# B&R Automation Studio project TD52 (part 101)

#### oilskidCyclic.st
```iecst
(*******************************************************************************
OilSkid	 				Oil Skid (cyclic)

This code is confidential AND proprietary to the INNIO Company.
It may NOT be used in any form, or reproduced in any manner,
without written permission of the INNIO Company.
Copyright, INNIO Company, 2019

Customized modifications: -
------------------------

History:
-------
V3.50	07.01.2014	Tinello 	created
		14.11.2014	Tinello		update TO NEW spezi
V4.x	05.12.2014	Walid Mari 	ported into XT4
V4.03.0	24.06.2015	lettenb.	bT_RelOilSkidPumpC: hy for oiltemp.limit circulation pump added
		18.09.2015				demand oilskid for N2 scavenging + ignition selftest added
		21.10.2015				xTOF_PrelubeDem: lag run time added
V4.05.0	04.04.2017	lettenb.	fast start added
V4.05.1	04.04.2018				bRelEngStart_OilSkid interface prepared for series
V4.05.2	25.04.2018	lettenb.	IN_GC.bOilskidDemSTFS demand for slowturn removed, SWAT920/5
V4.07.0 29.11.2018	lettenb.	preheating temp.limits 30/40->40/50°C
		12.02.2019	lettenb.	2505,3428,3431 depending on oil tank temp. OR oil supply temp.
								2508,3446 enable at engine shutdown
V4.07.1 08.04.2019				OUT_GC.tOilSkid_Heater.Do: bN_EngAct_IsZero removed, heater is active until set temp.is reached(krainz, alessio)
		30.07.2019	lettenb.	error condition for OilSkid: 1031 added, corr.for iCnt_OilSkid_HP_PrErr(safety request, doujak andreas) bu01
V4.10.0	03.08.2020	lettenb.	OUT_interfaces for op_state(bEng_Bloc) added
		14.12.2020	lettenb.	TON,TOF reset added to avoid time overrun, cleanup

Instructions FOR use:
--------------------

Description:
------------

Outstandings:
------------

(*******************************************************************************)
PROGRAM _CYCLIC

	(*----------------------------------------------*)
	(* RESET of alarms and warnings 				*)
	(*----------------------------------------------*)
	bAMM_Lev_OilSkid_Sump_Hi		:= FALSE;

	bAMM_Lev_OilSkid_Tank_Ms 		:= FALSE;
	bAMM_Lev_OilSkid_Tank_Lo 		:= FALSE;
	bAMM_Lev_OilSkid_Tank_LoLo 		:= FALSE;

	bAMM_T_OilSkid_Tank_Ms 			:= FALSE;
	bAMM_T_OilSkid_Tank_Lo 			:= FALSE;

	bAMM_T_OilSkid_Supply_Ms 		:= FALSE;
	bAMM_T_OilSkid_Supply_Lo 		:= FALSE;
	bAMM_T_OilSkid_Supply_Hi 		:= FALSE;

	bAMM_Flow_OilSkid_DE_Ms 		:= FALSE;
	bAMM_Flow_OilSkid_DE_Lo 		:= FALSE;
	bAMM_Flow_OilSkid_DE_Hi 		:= FALSE;

	bAMM_Flow_OilSkid_NDE_Ms 		:= FALSE;
	bAMM_Flow_OilSkid_NDE_Lo 		:= FALSE;
	bAMM_Flow_OilSkid_NDE_Hi 		:= FALSE;

	bAMM_Pr_OilSkid_HP_DE_Ms		:= FALSE;
	bAMM_Pr_OilSkid_HP_DE_Lo 		:= FALSE;

	bAMM_Pr_OilSkid_HP_NDE_Ms		:= FALSE;
	bAMM_Pr_OilSkid_HP_NDE_Lo 		:= FALSE;

	bAMM_OilSkid_PumpC_CB			:= FALSE;
	bAMM_DPr_OilSkid_FiltLP_Hi 		:= FALSE;
	bAMM_DPr_OilSkid_FiltHP_DE_Hi 	:= FALSE;
	bAMM_DPr_OilSkid_FiltHP_NDE_Hi 	:= FALSE;

	bAMM_OilSkid_PumpLP_CB 			:= FALSE;
	bAMM_OilSkid_PumpHP_CB 			:= FALSE;
	bAMM_OilSkid_PumpHP_CB_UPS 		:= FALSE;
	bAMM_OilSkid_Fan_CB 			:= FALSE;
	bAMM_OilSkid_Heater_CB 			:= FALSE;

	bAMM_OilSkid_MCB 				:= FALSE;
	bAMM_OilSkid_AuxV 				:= FALSE;
	bAMM_OilSkid_AuxV_UPS 			:= FALSE;

	(*----------------------------------------------*)
	(* RESET of IO's								*)
	(*----------------------------------------------*)
	OUT_GC.tOilSkid_Fan.Do			:= FALSE;
	OUT_GC.tOilSkid_Heater.Do		:= FALSE;
	OUT_GC.tOilSkid_PumpLP.Do		:= FALSE;
	OUT_GC.tOilSkid_PumpHP.Do		:= FALSE;
	OUT_GC.tOilSkid_PumpHP_UPS.Do	:= FALSE;
	OUT_GC.tOilSkid_PumpHP_Soft.Do	:= FALSE;
	OUT_GC.tOilSkid_PumpC.Do		:= FALSE;

	IF Para.bOilSkid_Exist AND IN_GC.tPB2MM.bParaSetupOk  THEN
		(****************************************************************************************************************************************)
		(* monitoring																															*)
		(****************************************************************************************************************************************)
		xTON_PumpLP_10s(IN:= MM2VIS.bOilSkid_PumpLP_Dem, PT:= T#10s); 								(* LP pump runs for 10 seconds *)
		xTON_PumpHP_5s(IN := MM2VIS.bOilSkid_PumpHP_Dem, PT:= T#5s); 								(* HP pump runs for 5 seconds *)

		(*----------------------------------------------*)
		(* error by DI									*)
		(*----------------------------------------------*)
		bAMM_Lev_OilSkid_Sump_Hi		:=  NOT IN_GC.tLev_OilSkid_Sump_Hi.Di; 										(* G.03-LS-001  *)	(* W3418 *)
		bAMM_DPr_OilSkid_FiltLP_Hi 		:=  NOT IN_GC.tDPr_OilSkid_FiltLP_Hi.Di										(* G.03-PDS-001 *)	(* W2505 *)
										AND 	xTON_PumpLP_10s.Q
										AND   ((bRelMon_T_Supply AND IN_GC.tT_OilSkid_Supply.Ai > 55) OR (bRelMon_T_Tank AND IN_GC.tT_OilSkid_Tank.Ai > 55));

		IF (IN_GC.rN_EngAct < 500 AND IN_GC.rN_EngAct > 100 AND NOT IN_GC.bEng_RPSDem) THEN
			bAMM_DPr_OilSkid_FiltHP_DE_Hi  := NOT IN_GC.tDPr_OilSkid_FiltHP_DE_Hi.Di  AND MM2VIS.bOilSkid_PumpHP_Dem;(* G.03-PDS-002 *) (* W2508 *)
			bAMM_DPr_OilSkid_FiltHP_NDE_Hi := NOT IN_GC.tDPr_OilSkid_FiltHP_NDE_Hi.Di AND MM2VIS.bOilSkid_PumpHP_Dem;(* G.03-PDS-003 *) (* W3446 *)
		END_IF;

		bAMM_OilSkid_PumpLP_CB 			:= NOT IN_GC.tOilSkid_PumpLP_CBOk.Di;															(* W3426 *)
		bAMM_OilSkid_PumpHP_CB 			:= NOT IN_GC.tOilSkid_PumpHP_CBOk.Di;															(* W3433 *)
		bAMM_OilSkid_PumpHP_CB_UPS 		:= NOT IN_GC.tOilSkid_PumpHP_CBOk_UPS.Di;														(* W3434 *)
		bAMM_OilSkid_Fan_CB 			:= NOT IN_GC.tOilSkid_Fan_CBOk.Di; 																(* W3437 *)
		bAMM_OilSkid_Heater_CB 			:= NOT IN_GC.tOilSkid_Heater_CBOk.Di;															(* W3438 *)
		bAMM_OilSkid_PumpC_CB			:= NOT IN_GC.tOilSkid_PumpC_CBOk.Di;															(* W3447 *)

		bAMM_OilSkid_MCB 				:= NOT IN_GC.tOilSkid_MCB.Di;																	(* W3439 *)
		bAMM_OilSkid_AuxV 				:= NOT IN_GC.tOilSkid_AuxV_Ok.Di		AND NOT bAMM_OilSkid_PumpHP_CB  						(* W3440 *)
																				AND NOT bAMM_OilSkid_MCB;
		bAMM_OilSkid_AuxV_UPS 			:= NOT IN_GC.tOilSkid_AuxV_Ok_UPS.Di	AND NOT bAMM_OilSkid_PumpHP_CB_UPS;						(* W3441 *)

			bErr_OilSkid_NoVoltage		:= bAMM_OilSkid_MCB OR bAMM_OilSkid_AuxV;

		(*----------------------------------------------*)
		(* error by measurement signal failure 			*)
		(*----------------------------------------------*)
		bAMM_Lev_OilSkid_Tank_Ms	:= Para.bLev_OilSkid_Tank_Exist 	AND NOT IN_GC.tLev_OilSkid_Tank.GoodQual;						(* W3419 *)
		bAMM_T_OilSkid_Tank_Ms		:= Para.bT_OilSkid_Tank_Exist 		AND NOT IN_GC.tT_OilSkid_Tank.GoodQual;							(* W3421 *)
		bAMM_T_OilSkid_Supply_Ms	:= Para.bT_OilSkid_Supply_Exist 	AND NOT IN_GC.tT_OilSkid_Supply.GoodQual;						(* W3423 *)
		bAMM_Flow_OilSkid_DE_Ms		:= Para.bFlow_OilSkid_DE_Exist 		AND NOT IN_GC.tFlow_OilSkid_DE.GoodQual;						(* W3427 *)
		bAMM_Flow_OilSkid_NDE_Ms	:= Para.bFlow_OilSkid_NDE_Exist 	AND NOT IN_GC.tFlow_OilSkid_NDE.GoodQual;						(* W3430 *)
		bAMM_Pr_OilSkid_HP_DE_Ms	:= Para.bPr_OilSkid_HP_DE_Exist 	AND NOT IN_GC.tPr_OilSkid_HP_DE.GoodQual;						(* W3435 *)
		bAMM_Pr_OilSkid_HP_NDE_Ms	:= Para.bPr_OilSkid_HP_NDE_Exist 	AND NOT IN_GC.tPr_OilSkid_HP_NDE.GoodQual;						(* W3442 *)

			(* Release monitoring	*)
			xTOF_AMM_Lev_Tank_Ms(IN := bAMM_Lev_OilSkid_Tank_Ms, 	PT:= T#10s);	(* TOF because of filtered signals *)
			xTOF_AMM_T_Tank_Ms(IN 	:= bAMM_T_OilSkid_Tank_Ms, 	 	PT:= T#10s);
			xTOF_AMM_T_Supply_Ms(IN := bAMM_T_OilSkid_Supply_Ms, 	PT:= T#10s);
			xTOF_AMM_Flow_DE_Ms(IN 	:= bAMM_Flow_OilSkid_DE_Ms, 	PT:= T#10s);
			xTOF_AMM_Flow_NDE_Ms(IN := bAMM_Flow_OilSkid_NDE_Ms, 	PT:= T#10s);
			xTOF_Pr_HP_DE_Ms(IN 	:= bAMM_Pr_OilSkid_HP_DE_Ms,	PT:= T#10s);
			xTOF_Pr_HP_NDE_Ms(IN 	:= bAMM_Pr_OilSkid_HP_NDE_Ms,	PT:= T#10s);

			bRelMon_Lev_Tank		:= Para.bLev_OilSkid_Tank_Exist		AND NOT xTOF_AMM_Lev_Tank_Ms.Q;
			bRelMon_T_Tank			:= Para.bT_OilSkid_Tank_Exist		AND NOT xTOF_AMM_T_Tank_Ms.Q;
			bRelMon_T_Supply		:= Para.bT_OilSkid_Supply_Exist		AND NOT xTOF_AMM_T_Supply_Ms.Q;
			bRelMon_Flow_DE			:= Para.bFlow_OilSkid_DE_Exist		AND NOT xTOF_AMM_Flow_DE_Ms.Q;
			bRelMon_Flow_NDE		:= Para.bFlow_OilSkid_NDE_Exist		AND NOT xTOF_AMM_Flow_NDE_Ms.Q;
			bRelMon_Pr_HP_DE		:= Para.bPr_OilSkid_HP_DE_Exist		AND NOT xTOF_Pr_HP_DE_Ms.Q;
			bRelMon_Pr_HP_NDE		:= Para.bPr_OilSkid_HP_NDE_Exist	AND NOT xTOF_Pr_HP_NDE_Ms.Q;

		(*----------------------------------------------*)
		(* error by level 		 						*)
		(*----------------------------------------------*)
		xGR_MINR_Lev_OilSkid_Tank(In:= IN_GC.tLev_OilSkid_Tank.Ai, Gw:= Para.rLev_OilSkid_Tank_LoLo, Hy:= 0.05);	(* 5% hysteresis *)

		bAMM_Lev_OilSkid_Tank_LoLo	:= xGR_MINR_Lev_OilSkid_Tank.Q 								AND bRelMon_Lev_Tank;					(* A2208 *)
		bAMM_Lev_OilSkid_Tank_Lo	:= (IN_GC.tLev_OilSkid_Tank.Ai < Para.rLev_OilSkid_Tank_Lo) AND bRelMon_Lev_Tank;					(* W3420 *)

		(*----------------------------------------------*)
		(* error by temperature	 						*)
		(*----------------------------------------------*)
		bAMM_T_OilSkid_Tank_Lo 		:= (IN_GC.tT_OilSkid_Tank.Ai   < 20) AND bOMSS_MAT AND bRelMon_T_Tank;								(* W3422 *)

		bAMM_T_OilSkid_Supply_Lo	:= (IN_GC.tT_OilSkid_Supply.Ai < Para.rT_OilSkid_Supply_Lo)	AND bRelMon_T_Supply					(* W3424 *)
																								AND MM2VIS.bOilSkid_PumpLP_Dem
																								AND bEng_Run_30m;

		bAMM_T_OilSkid_Supply_Hi	:= (IN_GC.tT_OilSkid_Supply.Ai > Para.rT_OilSkid_Supply_Hi)	AND bRelMon_T_Supply
																								AND MM2VIS.bOilSkid_PumpLP_Dem;			(* W3425 *)

		(*----------------------------------------------*)
		(* error by flow		 						*)
		(*----------------------------------------------*)
		IF (bRelMon_T_Supply AND IN_GC.tT_OilSkid_Supply.Ai > 55) OR 			(* tank   temperature > 55°C *)
		   (bRelMon_T_Tank   AND IN_GC.tT_OilSkid_Tank.Ai   > 55) THEN 			(* supply temperature > 55°C *)
			bErr_Flow_OilSkid_DE_Lo		:= (IN_GC.tFlow_OilSkid_DE.Ai  < Para.rFlow_OilSkid_DE_Lo);
			bErr_Flow_OilSkid_NDE_Lo	:= (IN_GC.tFlow_OilSkid_NDE.Ai < Para.rFlow_OilSkid_NDE_Lo);
		ELSE
			bErr_Flow_OilSkid_DE_Lo		:= (IN_GC.tFlow_OilSkid_DE.Ai  < 4);	(* 4 l/min *)
			bErr_Flow_OilSkid_NDE_Lo	:= (IN_GC.tFlow_OilSkid_NDE.Ai < 4);	(* 4 l/min *)
		END_IF;

		bAMM_Flow_OilSkid_DE_Lo		:= bErr_Flow_OilSkid_DE_Lo	AND xTON_PumpLP_10s.Q			AND bRelMon_Flow_DE;					(* W3428 *)
		bAMM_Flow_OilSkid_NDE_Lo	:= bErr_Flow_OilSkid_NDE_Lo	AND xTON_PumpLP_10s.Q			AND bRelMon_Flow_NDE;					(* W3431 *)

		bAMM_Flow_OilSkid_DE_Hi		:= (IN_GC.tFlow_OilSkid_DE.Ai  > Para.rFlow_OilSkid_DE_Hi)	AND bRelMon_Flow_DE;					(* W3429 *)
		bAMM_Flow_OilSkid_NDE_Hi	:= (IN_GC.tFlow_OilSkid_NDE.Ai > Para.rFlow_OilSkid_NDE_Hi)	AND bRelMon_Flow_NDE;					(* W3432 *)

		(*----------------------------------------------*)
		(* error by pressure	 						*)
		(*----------------------------------------------*)
			(* oil pressure in high pressure circuit OK *)
			bPr_OilSkid_HP_DE_Ok	:= IN_GC.tPr_OilSkid_HP_DE.Ai  > Para.rPr_OilSkid_HP_Lo;
			bPr_OilSkid_HP_NDE_Ok	:= IN_GC.tPr_OilSkid_HP_NDE.Ai > Para.rPr_OilSkid_HP_Lo;

			(* release by stable oil pressure *)
			xTON_PressOK_2s(IN:= ((bPr_OilSkid_HP_DE_Ok  AND bRelMon_Pr_HP_DE)  OR NOT Para.bPr_OilSkid_HP_DE_Exist ) AND
								 ((bPr_OilSkid_HP_NDE_Ok AND bRelMon_Pr_HP_NDE) OR NOT Para.bPr_OilSkid_HP_NDE_Exist) AND
								 (Para.bPr_OilSkid_HP_DE_Exist OR Para.bPr_OilSkid_HP_NDE_Exist),		(* at least on sensor exist *)
							PT:= T#2s);
			bRel_OilSkid_Pr	  := xTON_PressOK_2s.Q;

		bAMM_Pr_OilSkid_HP_DE_Lo 	:= NOT bPr_OilSkid_HP_DE_Ok	 AND xTON_PumpHP_5s.Q AND bRelMon_Pr_HP_DE;								(* W3436 *)
		bAMM_Pr_OilSkid_HP_NDE_Lo 	:= NOT bPr_OilSkid_HP_NDE_Ok AND xTON_PumpHP_5s.Q AND bRelMon_Pr_HP_NDE;							(* W3443 *)

		(****************************************************************************************************************************************)
		(* control																																*)
		(****************************************************************************************************************************************)
		xTOF_NoSpeed_30s(IN:= NOT bN_EngAct_IsZero, PT:= T#30s);							(* engine is running *)

			(*----------------------------------------------*)
			(* preheating		 							*)
			(*----------------------------------------------*)
			IF bRelMon_T_Tank AND bOMSS_MAT THEN
				IF 		IN_GC.tT_OilSkid_Tank.Ai >= 50 	THEN   bOilSkid_Heater	:= FALSE;
				ELSIF 	IN_GC.tT_OilSkid_Tank.Ai <  40 	THEN   bOilSkid_Heater	:= TRUE; 	END_IF;

				OUT_GC.tOilSkid_Heater.Do	:=	bOilSkid_Heater
										AND NOT bAMM_OilSkid_Heater_CB
										AND NOT bErr_OilSkid_NoVoltage
										AND NOT IN_GC.bMsg1031
										AND NOT IN_GC.bMsg1054;
			END_IF;

			(*----------------------------------------------*)
			(* Service										*)
			(*----------------------------------------------*)
			IF 		NOT M_DREHZ							(* engine is not running *)
				AND NOT bAMM_Lev_OilSkid_Sump_Hi
				AND NOT IN_GC.bEng_RPSDem				(* engine is not demanded *)
				AND    (IN_GC.tT_OilSkid_Tank.Ai >= 20) (* oil temperature OK *)
				AND     bRelMon_T_Tank  THEN

				(* oilskid oil high pressure pump runtime *)
				xTON_PumpHP_DemOn(IN:= bPumpHP_DemService, PT:= Para.tiOilSkid_PumpHP_Run);

				IF 	IN_GC.tOilSkid_PumpHP_DemOn.Di AND NOT xTOF_NoSpeed_30s.Q			THEN bPumpHP_DemService	:= TRUE; 	END_IF;
				IF (IN_GC.tOilSkid_PumpHP_DemOff.Di OR xTON_PumpHP_DemOn.Q) 			THEN bPumpHP_DemService	:= FALSE;	END_IF;

				(* reset if pump isn't running *)
				IF (xTON_PumpHP_DemOn.ET > T#5s) AND NOT MM2VIS.bOilSkid_PumpHP_Dem 	THEN bPumpHP_DemService	:= FALSE;	END_IF;

				(* demand oilskid oil high pressure pump for N2 or IgnSelfTest *)//SWAT920/5
				xTOF_PrelubeDem(IN:= IN_GC.bN2_ScavCoPrelubeOn OR IN_GC.bEO_PrelubeDemIgn, PT:= T#60s);(* lag run time / until engine stand still *)//SWAT920/5
				bPumpHP_DemN2Ign := xTOF_PrelubeDem.Q;

			ELSE
				xTON_PumpHP_DemOn(IN:= FALSE, PT:= T#0s);
				xTOF_PrelubeDem  (IN:= FALSE, PT:= T#0s);

				bPumpHP_DemService 	:= FALSE;
				bPumpHP_DemN2Ign	:= FALSE;
			END_IF;

			OUT_GC.bRelEngTurn_OilSkid	:= bRel_OilSkid_Pr AND(bPumpHP_DemService OR bPumpHP_DemN2Ign);	(* release engine turn *)

			(*----------------------------------------------*)
			(* release engine operation						*)
			(*----------------------------------------------*)
			IF    IN_GC.bEng_RPSDem AND (IN_GC.tT_OilSkid_Tank.Ai >= 20)
			THEN
				bPumpHP_DemEngOp			:= (IN_GC.rN_EngAct < 500);
				OUT_GC.tOilSkid_PumpLP.Do	:= (IN_GC.rN_EngAct > 200)
										AND NOT bAMM_OilSkid_PumpLP_CB
										AND NOT bErr_OilSkid_NoVoltage
										AND NOT IN_GC.bMsg1031
										AND NOT IN_GC.bMsg1054;
			ELSE
				bPumpHP_DemEngOp 		:= FALSE;
			END_IF;

			OUT_GC.bRelEngOp_OilSkid	:= bRel_OilSkid_Pr AND bPumpHP_DemEngOp;	(* release engine operation *)
			OUT_GC.bRelEngStart_OilSkid	:= NOT bAMM_T_OilSkid_Tank_Lo AND NOT bAMM_Lev_OilSkid_Tank_LoLo; (* oilskid ready for fast start *)

			(*----------------------------------------------*)
			(* cooling										*)
			(*----------------------------------------------*)
			IF NOT bN_EngAct_IsZero THEN

				IF 	bRelMon_T_Tank THEN
					IF 	  IN_GC.tT_OilSkid_Tank.Ai   >  Para.rT_OilSkid_Tank_Set 		THEN  bOilSkid_Fan	:= TRUE;
					ELSIF IN_GC.tT_OilSkid_Tank.Ai   < (Para.rT_OilSkid_Tank_Set - 5)	THEN  bOilSkid_Fan	:= FALSE; 	END_IF;

				ELSIF bRelMon_T_Supply 	THEN				(* switch to supply temperature in case of tank temp. error *)
					IF 	  IN_GC.tT_OilSkid_Supply.Ai >  Para.rT_OilSkid_Tank_Set 		THEN  bOilSkid_Fan	:= TRUE;
					ELSIF IN_GC.tT_OilSkid_Supply.Ai < (Para.rT_OilSkid_Tank_Set - 5) 	THEN  bOilSkid_Fan	:= FALSE; 	END_IF;
				END_IF;

				OUT_GC.tOilSkid_Fan.Do	:=	bOilSkid_Fan
									AND NOT bAMM_OilSkid_Fan_CB
									AND NOT bErr_OilSkid_NoVoltage
									AND NOT IN_GC.bMsg1031
									AND NOT IN_GC.bMsg1054;
			END_IF;

			(*----------------------------------------------*)
			(* circulation pump								*)
			(*----------------------------------------------*)
			IF 	  IN_GC.tT_OilSkid_Tank.Ai >= 22.0 THEN bT_RelOilSkidPumpC := TRUE;
			ELSIF IN_GC.tT_OilSkid_Tank.Ai <  20.0 THEN bT_RelOilSkidPumpC := FALSE; END_IF;

			OUT_GC.tOilSkid_PumpC.Do :=   ((MM2VIS.bOilSkid_Heater_Dem AND bT_RelOilSkidPumpC) OR (IN_GC.rN_EngAct > 200)) 	(* Heater is running *)
									AND	NOT bAMM_OilSkid_PumpC_CB
									AND NOT bErr_OilSkid_NoVoltage
									AND NOT IN_GC.bMsg1031
									AND NOT IN_GC.bMsg1054;

			(*----------------------------------------------*)
			(* engine stop									*)
			(*----------------------------------------------*)
			IF 	NOT IN_GC.bEng_RPSDem AND xTOF_NoSpeed_30s.Q THEN
				bPumpHP_DemEngStop			:= (IN_GC.rN_EngAct < 500);
				OUT_GC.tOilSkid_PumpLP.Do	:=	NOT bRel_OilSkid_Pr
											AND NOT bAMM_OilSkid_PumpLP_CB
											AND NOT bErr_OilSkid_NoVoltage
											AND NOT IN_GC.bMsg1031
											AND NOT IN_GC.bMsg1054;
				xTON_PumpHP_Dem_5s(IN := bPumpHP_DemEngStop, PT:= T#5s);	 			(* HP pump demand for 5 seconds *)

				IF  NOT bRel_OilSkid_Pr AND	EDGEPOS(xTON_PumpHP_Dem_5s.Q) THEN
					VIS2MM.iCnt_OilSkid_HP_PrErr := VIS2MM.iCnt_OilSkid_HP_PrErr + 1; 	(* Perm: error counter for high pressure *)
				END_IF;
			ELSE
				xTON_PumpHP_Dem_5s(IN:= FALSE, PT:= T#0s);
				bPumpHP_DemEngStop := FALSE;
			END_IF;

			(*----------------------------------------------*)
			(* engine faststart								*)
			(*----------------------------------------------*)
			xTON_FS(IN:= (IN_GC.rN_EngAct > 0), PT:= T#4s);
			IF 	IN_GC.bEng_Start THEN
				IF  NOT bRel_OilSkid_Pr AND	EDGEPOS(xTON_FS.Q) THEN
					VIS2MM.iCnt_OilSkid_HP_PrErr := VIS2MM.iCnt_OilSkid_HP_PrErr + 1; 	(* Perm: error counter for high pressure *)
				END_IF;
			END_IF;

			(*----------------------------------------------*)
			(* high pressure pump / UPS						*)
			(*----------------------------------------------*)
			xTOF_PumpHP_Dem(IN:= bPumpHP_DemService OR bPumpHP_DemN2Ign OR bPumpHP_DemEngOp OR bPumpHP_DemEngStop, PT:= T#1s);

			OUT_GC.tOilSkid_PumpHP_Soft.Do	:= xTOF_PumpHP_Dem.Q AND NOT IN_GC.bMsg1031
																 AND NOT IN_GC.bMsg1054;

			OUT_GC.tOilSkid_PumpHP.Do		:= xTOF_PumpHP_Dem.Q AND NOT xTOF_PumpHP_UPS.Q
																 AND NOT bAMM_OilSkid_PumpHP_CB
																 AND NOT bErr_OilSkid_NoVoltage
																 AND NOT IN_GC.bMsg1031
																 AND NOT IN_GC.bMsg1054;

			xTOF_PumpHP(IN:= OUT_GC.tOilSkid_PumpHP.Do, PT:= T#1s);

			OUT_GC.tOilSkid_PumpHP_UPS.Do	:= xTOF_PumpHP_Dem.Q AND NOT xTOF_PumpHP.Q
																 AND NOT bAMM_OilSkid_PumpHP_CB_UPS
																 AND NOT bAMM_OilSkid_AuxV_UPS
																 AND     xTOF_NoSpeed_30s.Q			(* demand only if shutdown *)
																 AND NOT IN_GC.bMsg1031
																 AND NOT IN_GC.bMsg1054;
			xTOF_PumpHP_UPS(IN:= OUT_GC.tOilSkid_PumpHP_UPS.Do, PT:= T#1s);

		IF 		IN_GC.bMsg1031  													(* A1031 emergency stop *)
			OR  IN_GC.bMsg1054  													(* A1054 fire alarm *)
			OR (MM2VIS.bMsg2208  AND NOT bMsg2208_Test) 							(* A2208 oilskid tank level minimum *)
			OR (bAMM_OilSkid_MCB AND     bN_EngAct_IsZero) THEN						(* W3439 Oilskid main switch auxiliaries opened *)

			bPumpHP_DemService 			:= FALSE;									(* NO demand of high pressure pump 	 *)
			bPumpHP_DemN2Ign			:= FALSE;									(* NO demand of high pressure pump 	 *)
			bPumpHP_DemEngOp			:= FALSE;									(* NO demand of high pressure pump 	 *)
			OUT_GC.bRelEngOp_OilSkid 	:= FALSE;									(* NO release of engine operation 	 *)
			OUT_GC.bRelEngTurn_OilSkid	:= FALSE;									(* NO release of engine barring gear *)
			OUT_GC.bRelEngStart_OilSkid	:= FALSE; 									(* NO oilskid ready for fast start   *)
		END_IF;

	ELSE (* inactive OilSkid *)
		xTON_PumpLP_10s(IN:= FALSE, PT:= T#0s);
		xTON_PumpHP_5s(IN:= FALSE, PT:= T#0s);
		xTON_PressOK_2s(IN:= FALSE, PT:= T#0s);
		xTON_PumpHP_DemOn(IN:= FALSE, PT:= T#0s);
		xTON_PumpHP_Dem_5s(IN:= FALSE, PT:= T#0s);
		xTON_FS(IN:= FALSE, PT:= T#0s);

		xTOF_NoSpeed_30s(IN:= FALSE, PT:= T#0s);
		xTOF_PrelubeDem(IN:= FALSE, PT:= T#0s);
		xTOF_PumpHP_UPS(IN:= FALSE, PT:= T#0s);
		xTOF_PumpHP(IN:= FALSE, PT:= T#0s);

		bPumpHP_DemService			:= FALSE;										(* NO demand of high pressure pump 	 *)
		bPumpHP_DemN2Ign			:= FALSE;										(* NO demand of high pressure pump 	 *)
		bPumpHP_DemEngOp			:= FALSE;										(* NO demand of high pressure pump 	 *)
		bPumpHP_DemEngStop			:= FALSE;										(* NO demand of high pressure pump 	 *)
		OUT_GC.bRelEngOp_OilSkid 	:= TRUE;										(*    release engine operation  	 *)
		OUT_GC.bRelEngTurn_OilSkid	:= TRUE;										(*    release engine barring gear	 *)
		OUT_GC.bRelEngStart_OilSkid	:= TRUE; 										(*    oilskid ready for fast start   *)
	END_IF;

	OUT_GC.bAMM_OilSkid_PumpLP_CB := bAMM_OilSkid_PumpLP_CB;						(* bEng_Bloc *)
	OUT_GC.bAMM_OilSkid_PumpHP_CB := bAMM_OilSkid_PumpHP_CB;						(* bEng_Bloc *)
	OUT_GC.bAMM_OilSkid_MCB       := bAMM_OilSkid_MCB;								(* bEng_Bloc *)

END_PROGRAM
```

#### oilskid.var
```iecst
VAR
	bErr_Flow_OilSkid_DE_Lo : BOOL := FALSE; (*Internal WARNING: OilSkid oil flow to DE - low*)
	bErr_Flow_OilSkid_NDE_Lo : BOOL := FALSE; (*Internal WARNING: OilSkid oil flow to NDE - low*)
	bErr_OilSkid_NoVoltage : BOOL := FALSE; (*Internal WARNING: OilSkid NO Voltage*)
	bOilSkid_Fan : BOOL := FALSE; (*Fan*)
	bOilSkid_Heater : BOOL := FALSE; (*Heater*)
	bPr_OilSkid_HP_DE_Ok : BOOL := FALSE; (*Oil pressure in high pressure circuit to DE bearing OK*)
	bPr_OilSkid_HP_NDE_Ok : BOOL := FALSE; (*Oil pressure in high pressure circuit to NDE bearing OK*)
	bPumpHP_DemEngOp : BOOL := FALSE; (*Demand high pressure pump for engine operation *)
	bPumpHP_DemEngStop : BOOL := FALSE; (*Demand high pressure pump for engine stop*)
	bPumpHP_DemService : BOOL := FALSE; (*Demand high pressure pump for service*)
	bPumpHP_DemN2Ign : BOOL := FALSE; (*Demand high pressure pump for N2 or IgnSelfTest*)
	bRelMon_Lev_Tank : BOOL := FALSE; (*Release monitoring OilSkid tank level*)
	bRelMon_Pr_HP_DE : BOOL := FALSE; (*Release monitoring OilSkid oil pressure in high pressure circuit to DE bearing*)
	bRelMon_Pr_HP_NDE : BOOL := FALSE; (*Release monitoring OilSkid oil pressure in high pressure circuit to NDE bearing*)
	bRelMon_T_Supply : BOOL := FALSE; (*Release monitoring OilSkid supply temperature*)
	bRelMon_T_Tank : BOOL := FALSE; (*Release monitoring OilSkid tank temperature*)
	bRel_OilSkid_Pr : BOOL := FALSE; (*Release by oil pressure*)
	bT_RelOilSkidPumpC : BOOL := FALSE; (*Release circ.pump by oil temperature*)
	xGR_MINR_Lev_OilSkid_Tank : GR_MINR := (0);
	xTOF_AMM_Flow_DE_Ms : TOF := (0);
	xTOF_AMM_Flow_NDE_Ms : TOF := (0);
	xTOF_AMM_Lev_Tank_Ms : TOF := (0);
	xTOF_AMM_T_Supply_Ms : TOF := (0);
	xTOF_AMM_T_Tank_Ms : TOF := (0);
	xTOF_NoSpeed_30s : TOF := (0);
	xTOF_Pr_HP_DE_Ms : TOF := (0);
	xTOF_Pr_HP_NDE_Ms : TOF := (0);
	xTOF_PumpHP : TOF := (0);
	xTOF_PumpHP_Dem : TOF := (0);
	xTOF_PumpHP_UPS : TOF := (0);
	xTON_PressOK_2s : TON := (0);
	xTON_PumpHP_5s : TON := (0);
	xTON_PumpHP_DemOn : TON := (0);
	xTON_PumpLP_10s : TON := (0);
	xTOF_PrelubeDem : TOF;
	xTON_FS : TON := (0);
	xTON_PumpHP_Dem_5s : TON := (0);
END_VAR
```

### Program Logical/Generator/PermGC (IEC, version 4.09.0) - + PermanentMemory

- PermGCCyclic.st (not readable text: treated as protected, skipped)

- PermGCInit.st (not readable text: treated as protected, skipped)

#### PermGC.var
```iecst
VAR
	pm_Error : UINT;
	write_once : BOOL;
	pm_len : UDINT;
	ModulName : STRING[35];
	DatObjInfo_01 : DatObjInfo;
	pm_id : UDINT;
	pm_p : UDINT;
	bCreateDataObj : BOOL;
	perm_par_vers : UINT;
	DatObjRead_01 : DatObjRead;
	DatObjDelete_PermMem : DatObjDelete;
	DatObjCreate_01 : DatObjCreate;
	DatObjWrite_01 : DatObjWrite;
	ulChecksumOld : UDINT;
	ulPMPointer : UDINT;
	ulChkValue : UDINT;
	TON_WritePMEM : TON;
	ulChecksum : UDINT;
	bWriteDataObj : BOOL;
	TON_WarnDelay : TON;
	TON_BlockMinFileAge : TON; (*waiting time without file write after successful performed write*)
	bBlock_MinFileAge : BOOL := FALSE; (*pause the perm file write after each sucessful write*)
	iPM_WriteCnt : UDINT; (* *) (*old VarName: usPMWriteCnt*)
END_VAR
VAR CONSTANT
	ERR_NOERROR : UINT := 0;
END_VAR
VAR
	pmm : Perm_GC_Struct;
END_VAR
```

### Program Logical/Generator/MsgGC (IEC, version 4.14.0) - messages

#### MsgGCCyclic.st
```iecst
(*******************************************************************************
MsgGC	 			 alarms generation MM_generator

This code is confidential and proprietary to the INNIO Company.
It may not be used in any form, or reproduced in any manner,
without written permission of the INNIO Company.
Copyright, INNIO Company, 2025

Customized modifications: -
------------------------

History:
-------
V0.01.0	02.11.2011	lettenb.	new
V0.01.0	22.04.2013	Denk		xMsg3319.Prio := 3; 	deleted (Copy-paste failure)
		27.05.2013	Lettenb.	reset OUT_xx.txx2AB.bGnlTripx changed
V0.02.0 21.06.2013	Zengerer	W3566 added
V4.00.0 04.03.2014	lettenb.	logger added
V4.00.1	19.05.2014	lettenb.	3566 bugfix
		30.05.2014				1037 prio4 -> 2, bugfix
V4.00.2	09.12.2014				1036.Enable := TRUE -> IN_GC.tPB2MM.bSys_Run(920 stapelfeld)
								1110 Aktivierung bei BR9 wenn n_nenn 20sec > 750rpm für (Einfahrprogramm 500rpm)(920 stapelfeld)
								1126,2277 bei BR9 nur aktiv wenn n_nenn > 750rpm	(wegen Einfahrprogramm)(920 stapelfeld)
								2202,2203,2204,2205,2206,2207,2502,2503,2504,2631,2632,2633,2634,2637 added (920)
V4.03.0	22.07.2015	lettenb.	1038,1073,1109,1110,1111,1112,1126,1127,1143,1144 modif. 2690,2691,3393 new, dyn.gridcode III(thaler)
								_TC2 var.removed(bugfix vvm maping failure)
V4.04.0	10.05.2016	lettenb.	1127 monitoring activation acc.specification(kru) removed(bU_Gen_Mon_Ena)
								3468 added(T_GenAirIn2)
		23.02.2017				3440 TON 2s hinzu, unterdrückung 3440 bei wiedereinschaltung hauptschalter/schutzschalter
		28.07.2017	502423184	A2202 AND A2203 disabled due TO SWAT 920 # 3
V4.05.0	06.12.2017	lettenb.	W3566 disabled(->3593/update gridcode functions)
								2316 added, 2277 bMMD_GenAlarmTestOn added, grid code logic(thaler)
		09.04.2018				1036 bParaSetupOk added to avoid alarm at plc startup, bugfix
V4.07.0	19.10.2018	lettenb.	3468 bParaSetupOk added to avoid alarm at plc startup, bugfix
		29.11.2018	lettenb.	2505 delay 10s->120s,3428 delay 120s, 3431 delay 120s, 2998 added
		15.02.2019	lettenb.	3429,3432 delay 0s->120s
		04.03.2019	lettenb.	1038,1144 IN_GC.tP_GenRev_Ext.Di / IN_GC.tI_GenAsy_Ext.Di - DIs act directly on alarms without delay
V4.07.1	04.06.2019	lettenb.	2336 added, 3573 disabled
V4.09.0	02.12.2019	lettenb.	9311 added, acc.VDE-AR-N 4110 / 10.2.3.1(thaler), protection test mapping
		03.02.2020	lettenb.	2156,2157,2998 write max.1x per minute, bugfix
		04.05.2020	lettenb.	xTON_SecTick added for cycle time undependency, bugfix
V4.10.0	22.12.2020	lettenb.	1112: RiskClass setting corr.acc.TI 1100-0111
V4.11.0	25.01.2020	MayerR		9285,9351 added, voltage droop, tU_SetExt_Norm -> tU_SetExtAI_Norm renamed
V4.12.0	21.11.2022	lettenb.	9365,9366,9367,9368 added, automatic bearing greasing system
								1109,1110: avoid alarm during gen.dexcitation and gcb closing to dead bb(DUB15 BF43),#912
		19.12.2022	Perktold	added comments for sr-code (EN 13849-1 / 4.6.3) for A1038
V4.13.0	12.06.2023	Rimal		2371 and 2372 added, oilskid
		04.07.2023	Perktold	A2373 and W9372 added, earth fault protection via MMD signals
V4.14.0	17.10.2024	Theobald	Alarm 1112,1121,1122,1123,1124,1125,1143,1144 priority changed from 2 to 3 (2024-223)
		25.10.2024	Farre		Reverse power status OUT_GC.bPact_Rev to SY (2024-241)
		18.11.2024	Farre		Enable "unbalance current monitoring A1144" based on Para.bCAsym_Ena (2024-234)
		04.03.2025	Perktold	Alarm 1144 priority changed back to 2 (from 3)

Instructions for use:
--------------------
1) declare alarm with function block "Alm"
	declare buffert alarm bit MM2VIS.bMsg<message number>

2) use template to create a new alarm,
   substitue 0000 by alarm number and make settings:

	xMsg0000.Enable		:=	TRUE;		enable/disable alarm
	xMsg0000.Set		:=	FALSE;		alarm set condition
	xMsg0000.PT			:=	T#0s;		alarm delay time
	xMsg0000.Prio		:=	1;			alarm priority: 1-3 = trip, 4 = warning
	xMsg0000.RiskClass	:=	3;			risk class for remote alarm reset
	xMsg0000.Reset		:=	FALSE;		FALSE: for all standard alarms	prio 1,2,3 and warnings prio 4
										TRUE : for autoreset alarms

	MM2VIS.bMsg0000			:=	xMsg0000.Q;	connect buffert alarm bit for VIS and control

3)  expand INIT

Outstandings:
------------
sort msg by number
(*******************************************************************************)
PROGRAM _CYCLIC

	(* reset general trip *)
	OUT_GC.tGC2AB.bGnlTrip1		:=	FALSE;
	OUT_GC.tGC2AB.bGnlTrip2		:=	FALSE;
	OUT_GC.tGC2AB.bGnlTrip3		:=	FALSE;
	OUT_GC.tGC2AB.bGnlWarning	:=	FALSE;
	OUT_GC.tGC2AB.bTriptype1	:=	FALSE;
	OUT_GC.tGC2AB.bTriptype2	:=	FALSE;
	OUT_GC.tGC2AB.bTriptype3	:=	FALSE;

	(*------------------------------------------------------------------------------*)
	xGR_MAX_M_D_1400(In := IN_GC.rN_EngAct,Gw := Para.rN_EngNom - 100.0, Hy := 10);
	M_D1400 := xGR_MAX_M_D_1400.Q AND IN_GC.tPB2MM.bParaSetupOk;

	xTON_FG_GENUW(IN := M_D1400 AND NOT IN_GC.tGenDeexitDem.Do, PT := T#20s);
	bU_Gen_Mon_Ena := xTON_FG_GENUW.Q;

	xTON_Eng_Run_10s(IN := IN_GC.tEng_Run.Do , PT := T#10s);
	bEng_Run_10s := xTON_Eng_Run_10s.Q;

	xTON_Eng_Run_20s(IN := IN_GC.tEng_Run.Do , PT := T#20s);
	bEng_Run_20s := xTON_Eng_Run_20s.Q;

	xGR_MAXR_M_HDREHZ(In := IN_GC.rN_EngAct , Gw := Para.rN_EngStart_LimHiHi, Hy := Para.rN_EngStart_HyHiHi );
	M_HDREHZ := xGR_MAXR_M_HDREHZ.Q AND IN_GC.tPB2MM.bParaSetupOk;

	xTON_AT24.IN := (IN_GC.tGCB_On.Di OR M_HDREHZ) AND (IN_GC.tEng_Run.Do OR (NOT IN_GC.tEng_SUExc_Rel.Di));
	xTON_AT24.PT := Para.tiP_Gen_Reverse;
	xTON_AT24();
	bP_Gen_Reverse := xTON_AT24.Q;

	xTP_RLSG_W.IN := IN_GC.bEng_Dem_EPS;
	xTP_RLSG_W.PT := Para.tiP_Reverse_Mon_Ena;
	xTP_RLSG_W();
	bP_Reverse_Mon_Ena := xTP_RLSG_W.Q;

	(* A1036 Generator overload/short circuit *)
	xMsg1036.Enable    := IN_GC.tPB2MM.bParaSetupOk;
	xMsg1036.Set       := NOT IN_GC.tOlShortCirc.Di;
	xMsg1036.PT        := T#0s;
	xMsg1036.RiskClass := 4;
	xMsg1036.Prio      := 2;
	xMsg1036.Reset     := FALSE;
	xMsg1036();
	OUT_GC.bMsg1036    := xMsg1036.Q;
	MM2VIS.bMsg1036    := xMsg1036.Q;

	(* A1037 generator winding temperature high (kaltleiter) *)
	xMsg1037.Enable    := NOT Para.bT_Gen_Wind_Ena;
	xMsg1037.Set       := bT_Gen_Wind_Max AND NOT MM2VIS.bMsg2105;
	xMsg1037.PT        := T#0s;
	xMsg1037.RiskClass := 4;
	xMsg1037.Prio      := 2;
	xMsg1037.Reset     := FALSE;
	xMsg1037();
	MM2VIS.bMsg1037    := xMsg1037.Q;

	(********************************************************************************************************************
	Safety-related application software source code (EN 13849-1 / 4.6.3): BEGIN
	*********************************************************************************************************************)

	(* A1038 Generator reverse power *)
	xTON_GSEIN(IN := IN_GC.tGCB_On.Di, PT := T#1m);
	SY_1m_rlsg := xTON_GSEIN.Q;

	xGR_MIN_AN_RLSG(In := IN_GC.rP_Act_Norm_Filt * IN_GC.rP_Nom, Gw := Para.rP_Reverse , Hy := Para.rP_Reverse_Hy);
	AN_RLSG := IN_GC.tPB2MM.bParaSetupOk AND xGR_MIN_AN_RLSG.Q;
	OUT_GC.bPact_Rev := AN_RLSG;

	IF IN_GC.bMMD_GenAlarmTestOn THEN	xTON_T28(IN:= AN_RLSG, PT:= Para.tiP_Gen_Reverse2);
	ELSE								xTON_T28(IN:= AN_RLSG AND bP_Gen_Reverse AND NOT bP_Reverse_Mon_Ena, PT:= Para.tiP_Gen_Reverse2);
	END_IF;

	T28 := xTON_T28.Q AND (NOT IN_GC.bSCO_Active OR NOT Para.bGlowIgnPrevActive);

	OUT_GC.bGCB_Off_RP := T28 AND (NOT MM2VIS.bMsg1038);

	(* Detect when GCB_Off_RP turns TRUE *)
	xR_TRIG_GCB_Off_RP(CLK := OUT_GC.bGCB_Off_RP);

	(* B3298 gcb opened by generator reverse power *)
	xTOF_GCB_Off_RP(IN := xR_TRIG_GCB_Off_RP.Q, PT:=T#10s);
	MM2VIS.bMsg3298 := xTOF_GCB_Off_RP.Q;

	xR_TRIG_T28(CLK := T28);

	IF xMsg1038.Q THEN
		xTP_RLSG2(IN := FALSE, PT := T#0s);
	ELSE
		xTP_RLSG2(IN := xR_TRIG_T28.Q AND RLSG1_arise, PT := T#60m);
	END_IF;

	RLSG2_arise := xTP_RLSG2.Q;

	IF xMsg1038.Q THEN
		xTP_RLSG1(IN := FALSE, PT := T#0s);
	ELSE
		xTP_RLSG1(IN := xR_TRIG_T28.Q, PT := T#60m);
	END_IF;

	RLSG1_arise := xTP_RLSG1.Q;

	xCTD_RLSG2(CD := T28, LOAD := NOT RLSG2_arise, PV := 3);
	xCTD_RLSG1(CD := T28, LOAD := NOT RLSG1_arise, PV := 3);
	STO_RLSG := xCTD_RLSG1.Q OR xCTD_RLSG2.Q;

	xMsg1038.Enable    := TRUE;
	xMsg1038.Set       := (T28 AND ((IN_GC.tGCB_On.Di AND (NOT IN_GC.tMCB_On.Di)) OR SY_1m_rlsg))
	                OR     STO_RLSG
					OR    (IN_GC.bMMD_GenAlarmTestOn AND xTON_T28.Q)
					OR NOT IN_GC.tP_GenRev_Ext.Di;
	xMsg1038.PT        := T#0s;
	xMsg1038.RiskClass := 10;
	xMsg1038.Prio      := 2;
	xMsg1038.Reset     := FALSE;
	xMsg1038();
	OUT_GC.bMsg1038    := xMsg1038.Q;
	MM2VIS.bMsg1038    := xMsg1038.Q;
	MM2VIS.bMsg1038Set := xMsg1038.Set;
	OUT_GC.bMsg1038Set := xMsg1038.Set;

	(********************************************************************************************************************
	Safety-related application software source code (EN 13849-1 / 4.6.3): END
	*********************************************************************************************************************)

	(* A1062 Measurement signal Excitation voltage (--> generally deactivated) *)
	xMsg1062.Enable    := FALSE;
	xMsg1062.Set       := NOT IN_GC.tU_Gen_Exc.GoodQual AND FALSE;
	xMsg1062.PT        := T#0s;
	xMsg1062.RiskClass := 4;
	xMsg1062.Prio      := 2;
	xMsg1062.Reset     := FALSE;
	xMsg1062();
	MM2VIS.bMsg1062    := xMsg1062.Q;

	(* A1073 Multi measurement device: generator overload/short circuit *)
	xMsg1073.Enable    := TRUE;
	xMsg1073.Set       := NOT IN_GC.tI_MMD_LimHi.Di;
	xMsg1073.PT        := T#0s;
	xMsg1073.RiskClass := 4;
	xMsg1073.Prio      := 2;
	xMsg1073.Reset     := FALSE;
	xMsg1073();
	OUT_GC.bMsg1073    := xMsg1073.Q;
	MM2VIS.bMsg1073    := xMsg1073.Q;

	(* A1109 generator loss of excitation *)
	xTOF_GenDeexitDem(IN:= IN_GC.tGenDeexitDem.Do, PT:= T#5s); (* no monitoring during generator deexcitation *)
	xTP_gcb_on2dead_bb(IN:= IN_GC.bGCB_aut_on2dead_bb, PT:= T#5s);

	xMsg1109.Enable    := TRUE;
	xMsg1109.Set       := NOT xTOF_GenDeexitDem.Q
                  AND     (bPF_CosPCtr_Trip         AND bP_Gen_Reverse AND NOT bP_Reverse_Mon_Ena)
					OR(NOT IN_GC.tGenLossExc_Ext.Di AND bP_Gen_Reverse AND NOT bP_Reverse_Mon_Ena)
					OR    (bPF_CosPCtr_Trip AND IN_GC.bMMD_GenAlarmTestOn);

	IF NOT xTP_gcb_on2dead_bb.Q THEN xMsg1109.PT := T#100ms;
	ELSE                        	 xMsg1109.PT := T#3s;
	END_IF;

	xMsg1109.RiskClass := 2;
	xMsg1109.Prio      := 2;
	xMsg1109.Reset     := FALSE;
	xMsg1109();
	MM2VIS.bMsg1109    := xMsg1109.Q;
	MM2VIS.bMsg1109Set := xMsg1109.Set;
	OUT_GC.bMsg1109Set := xMsg1109.Set;

	(* A1110 Generator frequency too low *)
	xTON_N_EngNom750(IN:= (Para.rN_EngNom > 750), PT:= T#20s);  // Deaktivierung für Einfahrprogramm BR9 500rpm
	xTON_Eng_Run_48s(IN:= IN_GC.tEng_Run.Do, PT:= T#48s);
	bEng_Run_48s := xTON_Eng_Run_48s.Q;

	xMsg1110.Enable    := TRUE;
	IF IN_GC.bMMD_GenAlarmTestOn THEN	xMsg1110.Set := NOT IN_GC.tF_MMD_LimLo[1].Di;
	ELSIF xEngType.Type9         THEN	xMsg1110.Set := NOT IN_GC.tF_MMD_LimLo[1].Di AND NOT xTOF_GenDeexitDem.Q AND bEng_Run_48s AND NOT bP_Reverse_Mon_Ena AND xTON_N_EngNom750.Q;
	ELSE								xMsg1110.Set := NOT IN_GC.tF_MMD_LimLo[1].Di AND NOT xTOF_GenDeexitDem.Q AND bEng_Run_20s AND NOT bP_Reverse_Mon_Ena;
	END_IF;

	IF NOT xTP_gcb_on2dead_bb.Q THEN xMsg1110.PT := T#100ms;
	ELSE                        	 xMsg1110.PT := T#3s;
	END_IF;

	xMsg1110.RiskClass := 1;
	xMsg1110.Prio      := 2;
	xMsg1110.Reset     := FALSE;
	xMsg1110();
	MM2VIS.bMsg1110    := xMsg1110.Q;
	MM2VIS.bMsg1110Set := xMsg1110.Set;
	OUT_GC.bMsg1110Set := xMsg1110.Set;

	(* A1111 Generator frequency too high *)
	xMsg1111.Enable    := TRUE;
	xMsg1111.Set       := (NOT IN_GC.tF_MMD_LimHi[1].Di AND bP_Gen_Reverse AND NOT bP_Reverse_Mon_Ena)
					   OR (NOT IN_GC.tF_MMD_LimHi[1].Di AND IN_GC.bMMD_GenAlarmTestOn);
	xMsg1111.PT        := T#0s;
	xMsg1111.RiskClass := 4;
	xMsg1111.Prio      := 2;
	xMsg1111.Reset     := FALSE;
	xMsg1111();
	MM2VIS.bMsg1111    := xMsg1111.Q;
	MM2VIS.bMsg1111Set := xMsg1111.Set;
	OUT_GC.bMsg1111Set := xMsg1111.Set;

	(* A1112 Neutral current maximum *)
	xMsg1112.Enable    := TRUE;
	xMsg1112.Set       := NOT IN_GC.tI_MMD_Neutr_LimHi[1].Di;
	xMsg1112.PT        := T#0s;
	xMsg1112.RiskClass := 2;
	xMsg1112.Prio      := 3;
	xMsg1112.Reset     := FALSE;
	xMsg1112();
	MM2VIS.bMsg1112    := xMsg1112.Q;
	MM2VIS.bMsg1112Set := xMsg1112.Set;
	OUT_GC.bMsg1112Set := xMsg1112.Set;

	(* A1113 Generator power measuring signal failure - for gen.power from Ai *)
	xMsg1113.Enable    := FALSE; (* true for mech.drive !!*)
	xMsg1113.Set       := NOT IN_GC.tP_Act[1].GoodQual AND bOMSS_Man AND NOT bP_Reverse_Mon_Ena;
	xMsg1113.PT        := T#1s;
	xMsg1113.RiskClass := 1;
	xMsg1113.Prio      := 2;
	xMsg1113.Reset     := FALSE;
	xMsg1113();
	MM2VIS.bMsg1113    := xMsg1113.Q;

	(* A1121 Generator winding temperature L1 Maximum *)
	xMsg1121.Enable    := Para.bT_Gen_Wind_Ena;
	xMsg1121.Set       := bT_Gen_Wind_L1_Max AND NOT MM2VIS.bMsg2106;
	xMsg1121.PT        := T#0s;
	xMsg1121.RiskClass := 4;
	xMsg1121.Prio      := 3;
	xMsg1121.Reset     := FALSE;
	xMsg1121();
	MM2VIS.bMsg1121    := xMsg1121.Q;

	(* A1122 Generator winding temperature L2 Maximum *)
	xMsg1122.Enable    := Para.bT_Gen_Wind_Ena;
	xMsg1122.Set       := bT_Gen_Wind_L2_Max AND NOT MM2VIS.bMsg2107;
	xMsg1122.PT        := T#0s;
	xMsg1122.RiskClass := 4;
	xMsg1122.Prio      := 3;
	xMsg1122.Reset     := FALSE;
	xMsg1122();
	MM2VIS.bMsg1122    := xMsg1122.Q;

	(* A1123 Generator winding temperature L3 Maximum *)
	xMsg1123.Enable    := Para.bT_Gen_Wind_Ena;
	xMsg1123.Set       := bT_Gen_Wind_L3_Max AND NOT MM2VIS.bMsg2108;
	xMsg1123.PT        := T#0s;
	xMsg1123.RiskClass := 4;
	xMsg1123.Prio      := 3;
	xMsg1123.Reset     := FALSE;
	xMsg1123();
	MM2VIS.bMsg1123    := xMsg1123.Q;

	(* A1124 Generator bearing temperature A maximum *)
	xMsg1124.Enable    := Para.bT_Gen_Bear_A_Ena;
	xMsg1124.Set       := bT_Gen_Bear_A_Max AND NOT MM2VIS.bMsg2109;
	xMsg1124.PT        := T#0s;
	xMsg1124.RiskClass := 4;
	xMsg1124.Prio      := 3;
	xMsg1124.Reset     := FALSE;
	xMsg1124();
	MM2VIS.bMsg1124    := xMsg1124.Q;

	(* A1125 Generator bearing temperature B maximum *)
	xMsg1125.Enable    := Para.bT_Gen_Bear_B_Ena;
	xMsg1125.Set       := bT_Gen_Bear_B_Max AND NOT MM2VIS.bMsg2110;
	xMsg1125.PT        := T#0s;
	xMsg1125.RiskClass := 4;
	xMsg1125.Prio      := 3;
	xMsg1125.Reset     := FALSE;
	xMsg1125();
	MM2VIS.bMsg1125    := xMsg1125.Q;

	(* A1126 Generator voltage low *)
	xMsg1126.Enable    := TRUE;
	IF IN_GC.bMMD_GenAlarmTestOn THEN	xMsg1126.Set := NOT IN_GC.tU_Gen_LimLo[1].Di;
	ELSIF xEngType.Type9 		 THEN	xMsg1126.Set := NOT IN_GC.tU_Gen_LimLo[1].Di AND bU_Gen_Mon_Ena AND(Para.rN_EngNom > 750);// Deaktivierung für Einfahrprogramm BR9 500rpm
	ELSE								xMsg1126.Set := NOT IN_GC.tU_Gen_LimLo[1].Di AND bU_Gen_Mon_Ena;
	END_IF;
	xMsg1126.PT        := T#0s;
	xMsg1126.RiskClass := 4;
	xMsg1126.Prio      := 2;
	xMsg1126.Reset     := FALSE;
	xMsg1126();
	MM2VIS.bMsg1126    := xMsg1126.Q;
	MM2VIS.bMsg1126Set := xMsg1126.Set;
	OUT_GC.bMsg1126Set := xMsg1126.Set;

	(* A1127 Generator voltage high *)
	xMsg1127.Enable    := TRUE;
	xMsg1127.Set       :=  NOT IN_GC.tU_Gen_LimHi[1].Di;
	xMsg1127.PT        := T#0s;
	xMsg1127.RiskClass := 4;
	xMsg1127.Prio      := 2;
	xMsg1127.Reset     := FALSE;
	xMsg1127();
	MM2VIS.bMsg1127    := xMsg1127.Q;
	MM2VIS.bMsg1127Set := xMsg1127.Set;
	OUT_GC.bMsg1127Set := xMsg1127.Set;

	(* A1132 Differential protection *)
	xSR_FG_DIFFUW(SET1  := M_D1400,
				  RESET := IN_GC.bEng_Start OR (NOT M_D1400 AND NOT IN_GC.bGV_On AND NOT IN_GC.bEng_Dem AND NOT IN_GC.tGCB_On.Di));
	xMsg1132.Enable    := TRUE;
	xMsg1132.Set       := NOT IN_GC.tDiffPrct.Di AND (xSR_FG_DIFFUW.Q1  OR (NOT Para.bPF_CosPCtr_Diff_Ena));
	xMsg1132.PT        := T#0s;
	xMsg1132.RiskClass := 4;
	xMsg1132.Prio      := 2;
	xMsg1132.Reset     := FALSE;
	xMsg1132();
	OUT_GC.bMsg1132    := xMsg1132.Q;
	MM2VIS.bMsg1132    := xMsg1132.Q;

	(* A1134 Earth failure generator *)(* W9311 *)
	xMsg1134.Enable    := TRUE;
	xMsg1134.Set       := NOT IN_GC.tGndFailure.Di;
	xMsg1134.PT        := T#0s;
	xMsg1134.RiskClass := 4;
	xMsg1134.Prio      := 2;
	xMsg1134.Reset     := FALSE;
	xMsg1134();
	OUT_GC.bMsg1134    := xMsg1134.Q;
	MM2VIS.bMsg1134    := xMsg1134.Q;

	(* A1143 Voltage negative sequence *)
	xGR_MAXR_DREHZ(In := IN_GC.rN_EngAct, Gw := 0.933 * Para.rN_EngNom, Hy := 0.0);
	FG_UASY := IN_GC.tEng_Run.Do AND xGR_MAXR_DREHZ.Q;

	xTON_UASY    (IN := NOT IN_GC.tU_MMD_Asy[1].Di AND FG_UASY,PT := T#3s);
	xTON_UASY_Ext(IN := NOT IN_GC.tU_GenAsy_Ext.Di AND FG_UASY,PT := T#3s);

	xMsg1143.Enable    := TRUE;
	xMsg1143.Set       := (NOT IN_GC.tU_MMD_Asy[1].Di AND FG_UASY AND xTON_UASY.Q)
					   OR (NOT IN_GC.tU_GenAsy_Ext.Di AND FG_UASY AND xTON_UASY_Ext.Q)
					   OR (NOT IN_GC.tU_MMD_Asy[1].Di AND IN_GC.bMMD_GenAlarmTestOn);
 	xMsg1143.PT        := T#0s;
	xMsg1143.RiskClass := 4;
	xMsg1143.Prio      := 3;
	xMsg1143.Reset     := FALSE;
	xMsg1143();
	MM2VIS.bMsg1143    := xMsg1143.Q;
	MM2VIS.bMsg1143Set := xMsg1143.Set;
	OUT_GC.bMsg1143Set := xMsg1143.Set;

	(* A1144 Current negative sequence *)
	xTON_GSEIN(IN := IN_GC.tGCB_On.Di , PT := T#1m);
	SY_1m_iasy          := xTON_GSEIN.Q;

	bIASY               := (NOT IN_GC.tI_MMD_Asy[1].Di  AND bEng_Run_10s);
	OUT_GC.bGCB_Off_CNS := Para.bCAsym_Ena AND bIASY AND (NOT MM2VIS.bMsg1144);

	(* Detect when GCB_Off_CNS turns TRUE *)
	xR_TRIG_GCB_Off_CNS(CLK := OUT_GC.bGCB_Off_CNS);

	(* B3299 Generator circuit breaker opened by current negative sequence *)
	xTOF_GCB_Off_CNS(IN := xR_TRIG_GCB_Off_CNS.Q, PT := T#10s);
	MM2VIS.bMsg3299 := xTOF_GCB_Off_CNS.Q;

	xR_TRIG_bIASY(CLK := bIASY);
	IF xMsg1144.Q THEN
		xTP_IASY2(IN := FALSE, PT := T#0s);
	ELSE
		xTP_IASY2(IN := xR_TRIG_bIASY.Q AND IASY1_arise, PT := T#60m);
	END_IF;

	IASY2_arise := xTP_IASY2.Q;

	IF xMsg1144.Q THEN
		xTP_IASY1(IN := FALSE, PT := T#0s);
	ELSE
		xTP_IASY1(IN := xR_TRIG_bIASY.Q, PT := T#60m);
	END_IF;

	IASY1_arise := xTP_IASY1.Q;

	xCTD_IASY1(CD := bIASY, LOAD := NOT IASY1_arise, PV := 3);
	xCTD_IASY2(CD := bIASY, LOAD := NOT IASY2_arise, PV := 3);
	STO_IASY      := xCTD_IASY1.Q OR xCTD_IASY2.Q;

	xMsg1144.Enable := TRUE;
	xMsg1144.Set    := Para.bCAsym_Ena
						AND ((bIASY AND ((IN_GC.tGCB_On.Di AND NOT IN_GC.tMCB_On.Di) OR SY_1m_iasy))
							OR  STO_IASY
							OR (NOT IN_GC.tI_MMD_Asy[1].Di AND IN_GC.bMMD_GenAlarmTestOn)
							OR  NOT IN_GC.tI_GenAsy_Ext.Di);
	xMsg1144.PT        := T#0s;
	xMsg1144.RiskClass := 4;
	xMsg1144.Prio      := 2;
	xMsg1144.Reset     := FALSE;
	xMsg1144();
	MM2VIS.bMsg1144    := xMsg1144.Q;
	MM2VIS.bMsg1144Set := xMsg1144.Set;
	OUT_GC.bMsg1144Set := xMsg1144.Set;

	(* W1154 Winding temperature L1 maximum *)
	xMsg1154.Enable    := Para.bT_Gen_Wind_Ena;
	xMsg1154.Set       := bT_Gen_Wind_L1_Lim AND NOT MM2VIS.bMsg2106;
	xMsg1154.PT        := T#0s;
	xMsg1154.RiskClass := 4;
	xMsg1154.Prio      := 4;
	xMsg1154.Reset     := FALSE;
	xMsg1154();
	MM2VIS.bMsg1154    := xMsg1154.Q;

	(* W1155 Winding temperature L2 maximum *)
	xMsg1155.Enable    := Para.bT_Gen_Wind_Ena;
	xMsg1155.Set       := bT_Gen_Wind_L2_Lim AND NOT MM2VIS.bMsg2107;
	xMsg1155.PT        := T#0s;
	xMsg1155.RiskClass := 4;
	xMsg1155.Prio      := 4;
	xMsg1155.Reset     := FALSE;
	xMsg1155();
	MM2VIS.bMsg1155    := xMsg1155.Q;

	(* W1156 Winding temperature L3 maximum *)
	xMsg1156.Enable    := Para.bT_Gen_Wind_Ena;
	xMsg1156.Set       := bT_Gen_Wind_L3_Lim AND NOT MM2VIS.bMsg2108;
	xMsg1156.PT        := T#0s;
	xMsg1156.RiskClass := 4;
	xMsg1156.Prio      := 4;
	xMsg1156.Reset     := FALSE;
	xMsg1156();
	MM2VIS.bMsg1156    := xMsg1156.Q;

	(* W1157 Bearing temperature A maximum *)
	xMsg1157.Enable    := Para.bT_Gen_Bear_A_Ena;
	xMsg1157.Set       := bT_Gen_Bear_A_Lim AND NOT MM2VIS.bMsg2109;
	xMsg1157.PT        := T#0s;
	xMsg1157.RiskClass := 4;
	xMsg1157.Prio      := 4;
	xMsg1157.Reset     := FALSE;
	xMsg1157();
	MM2VIS.bMsg1157    := xMsg1157.Q;

	(* W1158 Bearing temperature B maximum *)
	xMsg1158.Enable    := Para.bT_Gen_Bear_B_Ena;
	xMsg1158.Set       := bT_Gen_Bear_B_Lim AND NOT MM2VIS.bMsg2110;
	xMsg1158.PT        := T#0s;
	xMsg1158.RiskClass := 4;
	xMsg1158.Prio      := 4;
	xMsg1158.Reset     := FALSE;
	xMsg1158();
	MM2VIS.bMsg1158    := xMsg1158.Q;

	(* W1185 Winding temperature maximum *)
	xMsg1185.Enable    := NOT Para.bT_Gen_Wind_Ena;
	xMsg1185.Set       := bT_Gen_Wind_Lim AND NOT MM2VIS.bMsg2105;
	xMsg1185.PT        := T#0s;
	xMsg1185.RiskClass := 4;
	xMsg1185.Prio      := 4;
	xMsg1185.Reset     := FALSE;
	xMsg1185();
	MM2VIS.bMsg1185    := xMsg1185.Q;

	(* W2100 Differential protection relay failure *)
	xMsg2100.Enable    := TRUE;
	xMsg2100.Set       := NOT IN_GC.tI_Diff.Di;
	xMsg2100.PT        := T#0s;
	xMsg2100.RiskClass := 4;
	xMsg2100.Prio      := 4;
	xMsg2100.Reset     := FALSE;
	xMsg2100();
	MM2VIS.bMsg2100    := xMsg2100.Q;

	(* W2105 Measurement signal Generator winding temperature *)
	xMsg2105.Enable    := NOT Para.bT_Gen_Wind_Ena;
	xMsg2105.Set       := NOT IN_GC.tT_Gen_Wind.GoodQual AND IN_GC.tPB2MM.bParaSetupOk;
	xMsg2105.PT        := T#0s;
	xMsg2105.RiskClass := 4;
	xMsg2105.Prio      := 4;
	xMsg2105.Reset     := FALSE;
	xMsg2105();
	MM2VIS.bMsg2105    := xMsg2105.Q;

	(* W2106 Measurement signal Generator winding temperature L1 *)
	xMsg2106.Enable    := Para.bT_Gen_Wind_Ena;
	xMsg2106.Set       := NOT IN_GC.tT_Gen_Wind_Act_L1.GoodQual AND IN_GC.tPB2MM.bParaSetupOk;
	xMsg2106.PT        := T#0s;
	xMsg2106.RiskClass := 4;
	xMsg2106.Prio      := 4;
	xMsg2106.Reset     := FALSE;
	xMsg2106();
	MM2VIS.bMsg2106    := xMsg2106.Q;

	(* W2107 Measurement signal Generator winding temperature L2 *)
	xMsg2107.Enable    := Para.bT_Gen_Wind_Ena;
	xMsg2107.Set       := NOT IN_GC.tT_Gen_Wind_Act_L2.GoodQual AND IN_GC.tPB2MM.bParaSetupOk;
	xMsg2107.PT        := T#0s;
	xMsg2107.RiskClass := 4;
	xMsg2107.Prio      := 4;
	xMsg2107.Reset     := FALSE;
	xMsg2107();
	MM2VIS.bMsg2107    := xMsg2107.Q;

	(* W2108 Measurement signal Generator winding temperature L3 *)
	xMsg2108.Enable    := Para.bT_Gen_Wind_Ena;
	xMsg2108.Set       := NOT IN_GC.tT_Gen_Wind_Act_L3.GoodQual AND IN_GC.tPB2MM.bParaSetupOk;
	xMsg2108.PT        := T#0s;
	xMsg2108.RiskClass := 4;
	xMsg2108.Prio      := 4;
	xMsg2108.Reset     := FALSE;
	xMsg2108();
	MM2VIS.bMsg2108    := xMsg2108.Q;

	(* W2109 Measurement signal Generator bearing A temperature *)
	xMsg2109.Enable    := Para.bT_Gen_Bear_A_Ena;
	xMsg2109.Set       := NOT IN_GC.tT_Gen_Bear_A_Act.GoodQual AND IN_GC.tPB2MM.bParaSetupOk;
	xMsg2109.PT        := T#0s;
	xMsg2109.RiskClass := 4;
	xMsg2109.Prio      := 4;
	xMsg2109.Reset     := FALSE;
	xMsg2109();
	MM2VIS.bMsg2109    := xMsg2109.Q;

	(* W2110 Measurement signal Generator bearing B temperature *)
	xMsg2110.Enable    := Para.bT_Gen_Bear_B_Ena;
	xMsg2110.Set       := NOT IN_GC.tT_Gen_Bear_B_Act.GoodQual AND IN_GC.tPB2MM.bParaSetupOk;
	xMsg2110.PT        := T#0s;
	xMsg2110.RiskClass := 4;
	xMsg2110.Prio      := 4;
	xMsg2110.Reset     := FALSE;
	xMsg2110();
	MM2VIS.bMsg2110    := xMsg2110.Q;

	(* W2115 Generator voltage regulator failure *)
	xTON_GENREG_F(IN := ((    IN_GC.tU_Gen_Contr_Fail.Di AND NOT Para.bU_Gen_Contr_Sel) OR
	                     (NOT IN_GC.tU_Gen_Contr_Fail.Di AND     Para.bU_Gen_Contr_Sel)) , PT := Para.ti_Gen_VoltReg_Fail);
	ZM_GENREG_F        := xTON_GENREG_F.Q;

	xMsg2115.Enable    := TRUE;
	xMsg2115.Set       := ZM_GENREG_F AND bEng_Run_10s;
	xMsg2115.PT        := T#0s;
	xMsg2115.RiskClass := 4;
	xMsg2115.Prio      := 4;
	xMsg2115.Reset     := FALSE;
	xMsg2115();
	MM2VIS.bMsg2115    :=  xMsg2115.Q;

	(*  2202 generator DE bearing displacement trip *)
	xGR_MAX_F_GenBearDE1_HiHi(In:= IN_GC.tF_GenBear_DE1.Ai, Gw:= Para.rF_GenBear_HiHi, Hy:= 0.0);
	xGR_MAX_F_GenBearDE2_HiHi(In:= IN_GC.tF_GenBear_DE2.Ai, Gw:= Para.rF_GenBear_HiHi, Hy:= 0.0);

	xMsg2202.Enable    := FALSE; //SWAT920#3;
	xMsg2202.Set       := (xGR_MAX_F_GenBearDE1_HiHi.Q AND IN_GC.tF_GenBear_DE1.GoodQual)
					   OR (xGR_MAX_F_GenBearDE2_HiHi.Q AND IN_GC.tF_GenBear_DE2.GoodQual);
	xMsg2202.PT        := Para.tiF_GenBear_HiHi;
	xMsg2202.RiskClass := 4;
	xMsg2202.Prio      := 3;
	xMsg2202.Reset     := FALSE;
	xMsg2202();
	MM2VIS.bMsg2202    := xMsg2202.Q;

	(*  2203 generator NDE bearing displacement trip *)
	xGR_MAX_F_GenBearNDE1_HiHi(In:= IN_GC.tF_GenBear_NDE1.Ai, Gw:= Para.rF_GenBear_HiHi, Hy:= 0.0);
	xGR_MAX_F_GenBearNDE2_HiHi(In:= IN_GC.tF_GenBear_NDE2.Ai, Gw:= Para.rF_GenBear_HiHi, Hy:= 0.0);

	xMsg2203.Enable    := FALSE; //SWAT920#3;
	xMsg2203.Set       := (xGR_MAX_F_GenBearNDE1_HiHi.Q AND IN_GC.tF_GenBear_NDE1.GoodQual)
					   OR (xGR_MAX_F_GenBearNDE2_HiHi.Q AND IN_GC.tF_GenBear_NDE2.GoodQual);
	xMsg2203.PT        := Para.tiF_GenBear_HiHi;
	xMsg2203.RiskClass := 4;
	xMsg2203.Prio      := 3;
	xMsg2203.Reset     := FALSE;
	xMsg2203();
	MM2VIS.bMsg2203    := xMsg2203.Q;

	(*  2204 measuring signal failure displacement sensor 1 generator DE bearing (W2631) *)
	xMsg2204.Enable    := IN_GC.tPB2MM.bParaSetupOk	AND Para.bF_GenBear_DE1_Active AND FALSE;
	xMsg2204.Set       := NOT IN_GC.tF_GenBear_DE1.GoodQual;
	xMsg2204.PT        := T#0s;
	xMsg2204.RiskClass := 4;
	xMsg2204.Prio      := 3;
	xMsg2204.Reset     := FALSE;
	xMsg2204();
	MM2VIS.bMsg2204    :=  xMsg2204.Q;

	(*  2205 measuring signal failure displacement sensor 2 generator DE bearing (W2632) *)
	xMsg2205.Enable    := IN_GC.tPB2MM.bParaSetupOk	AND Para.bF_GenBear_DE2_Active AND FALSE;
	xMsg2205.Set       := NOT IN_GC.tF_GenBear_DE2.GoodQual;
	xMsg2205.PT        := T#0s;
	xMsg2205.RiskClass := 4;
	xMsg2205.Prio      := 3;
	xMsg2205.Reset     := FALSE;
	xMsg2205();
	MM2VIS.bMsg2205    :=  xMsg2205.Q;

	(*  2206 measuring signal failure displacement sensor 1 generator NDE bearing (W2633) *)
	xMsg2206.Enable    := IN_GC.tPB2MM.bParaSetupOk	AND Para.bF_GenBear_NDE1_Active AND FALSE;
	xMsg2206.Set       := NOT IN_GC.tF_GenBear_NDE1.GoodQual;
	xMsg2206.PT        := T#0s;
	xMsg2206.RiskClass := 4;
	xMsg2206.Prio      := 3;
	xMsg2206.Reset     := FALSE;
	xMsg2206();
	MM2VIS.bMsg2206    :=  xMsg2206.Q;

	(*  2207 measuring signal failure displacement sensor 2 generator NDE bearing (W2634) *)
	xMsg2207.Enable    := IN_GC.tPB2MM.bParaSetupOk	AND Para.bF_GenBear_NDE2_Active AND FALSE;
	xMsg2207.Set       := NOT IN_GC.tF_GenBear_NDE2.GoodQual;
	xMsg2207.PT        := T#0s;
	xMsg2207.RiskClass := 4;
	xMsg2207.Prio      := 3;
	xMsg2207.Reset     := FALSE;
	xMsg2207();
	MM2VIS.bMsg2207    :=  xMsg2207.Q;

	(* A2208 Oilskid tank oil level low *)
	xMsg2208.Enable		:= TRUE;
	xMsg2208.Set		:= bAMM_Lev_OilSkid_Tank_LoLo;
	xMsg2208.PT			:= T#0s;
	xMsg2208.Prio		:= 3;
	xMsg2208.Reset		:= FALSE;
	xMsg2208();
	MM2VIS.bMsg2208 	:= xMsg2208.Q;
	bMsg2208_Test		:= xMsg2208.Test;

	MM2VIS.bMsg2209; (*  2209 generator LOS oil outlet pressure low *)	(* --> NOT USED *)
	MM2VIS.bMsg2210; (*  2210 generator both LOS AC oil pumps failed *)	(* --> NOT USED *)
	MM2VIS.bMsg2211; (*  2211 generator LOS oil temperature high *)		(* --> NOT USED *)
	MM2VIS.bMsg2212; (*  2212 generator both JOS AC oil pumps failed *)	(* --> NOT USED *)
	MM2VIS.bMsg2213; (*  2213 ? *)	(* --> NOT USED *)
	MM2VIS.bMsg2235; (*  2235 ? *)	(* --> NOT USED *)

	(* A2277 Generator voltage too low 2*)
	xMsg2277.Enable    := TRUE;
	IF IN_GC.bMMD_GenAlarmTestOn THEN xMsg2277.Set := NOT IN_GC.tU_Gen_LimLo2[1].Di;
	ELSIF xEngType.Type9         THEN xMsg2277.Set := NOT IN_GC.tU_Gen_LimLo2[1].Di AND bU_Gen_Mon_Ena AND(Para.rN_EngNom > 750);// Deaktivierung für Einfahrprogramm BR9 500rpm
	ELSE		                      xMsg2277.Set := NOT IN_GC.tU_Gen_LimLo2[1].Di AND bU_Gen_Mon_Ena;
	END_IF;
	xMsg2277.PT        := T#0s;
	xMsg2277.RiskClass := 4;
	xMsg2277.Prio      := 2;
	xMsg2277.Reset     := FALSE;
	xMsg2277();
	MM2VIS.bMsg2277    := xMsg2277.Q;
	MM2VIS.bMsg2277Set := xMsg2277.Set;
	OUT_GC.bMsg2277Set := xMsg2277.Set;

	(* A2316 Generator voltage high 2 *)
	xMsg2316.Enable    := TRUE;
	xTON2316Set(IN:=   (IN_GC.tU_L1L2[1].Ai >= Para.rU_Gen_Nom[1] * Para.rV_Over2[1])
					OR (IN_GC.tU_L2L3[1].Ai >= Para.rU_Gen_Nom[1] * Para.rV_Over2[1])
					OR (IN_GC.tU_L3L1[1].Ai >= Para.rU_Gen_Nom[1] * Para.rV_Over2[1]),
				PT:= REAL_TO_TIME(Para.rTi_V_Over2[1] * 1000));
	xMsg2316.Set       := xTON2316Set.Q;
	xMsg2316.PT        := T#0s;
	xMsg2316.RiskClass := 4;
	xMsg2316.Prio      := 2;
	xMsg2316.Reset     := FALSE;
	xMsg2316();
	MM2VIS.bMsg2316    := xMsg2316.Q;
	MM2VIS.bMsg2316Set := xMsg2316.Set;
	OUT_GC.bMsg2316Set := xMsg2316.Set;

	(* A2336 Failure Generator lubricating oil - Cooling *)
	xMsg2336.Enable    := TRUE;
	xMsg2336.Set       := NOT IN_GC.tGen_LO_CoolingSys_Fail.Di;
	xMsg2336.PT        := T#0s;
	xMsg2336.RiskClass := 4;
	xMsg2336.Prio      := 3;
	xMsg2336.Reset     := FALSE;
	xMsg2336();
	MM2VIS.bMsg2336    := xMsg2336.Q;

	(* A2371 Oil skid Oil flow to DE bearing Low *)
	xMsg2371.Enable    := TRUE;
	xMsg2371.Set       := (IN_GC.tFlow_OilSkid_DE.Ai < 2.0) AND (IN_GC.rN_EngAct > 500) AND bRelMon_Flow_DE;
	xMsg2371.PT        := T#60s;
	xMsg2371.RiskClass := 4;
	xMsg2371.Prio      := 3;
	xMsg2371.Reset     := FALSE;
	xMsg2371();
	MM2VIS.bMsg2371    := xMsg2371.Q;

	(* A2372 Oil skid Oil flow to NDE bearing Low *)
	xMsg2372.Enable    := TRUE;
	xMsg2372.Set       := (IN_GC.tFlow_OilSkid_NDE.Ai < 2.0) AND (IN_GC.rN_EngAct > 500) AND bRelMon_Flow_NDE;
	xMsg2372.PT        := T#60s;
	xMsg2372.RiskClass := 4;
	xMsg2372.Prio      := 3;
	xMsg2372.Reset     := FALSE;
	xMsg2372();
	MM2VIS.bMsg2372    := xMsg2372.Q;

	(* A2373 Earth failure generator (MMD) *)
	xMsg2373.Enable	:= 	NOT IN_GC.bSimWinMOD_Active;
	xMsg2373.Set 	:=	bMsg2373_set;
	xMsg2373.PT 	:=	T#0s;
	xMsg2373.Prio	:= 	2;
	xMsg2373.Reset	:= 	FALSE;
	xMsg2373();
	MM2VIS.bMsg2373	:= xMsg2373.Q;

	(* W2501 Generator rotating diode failure *)
	xMsg2501.Enable    := TRUE;
	xMsg2501.Set       :=(IN_GC.tU_GenDiode_Fail.Di OR IN_GC.tU_GenDiode_Trip.Di) AND bEng_Run_10s;
	xMsg2501.PT        := T#5s;
	xMsg2501.RiskClass := 4;
	xMsg2501.Prio      := 4;
	xMsg2501.Reset     := FALSE;
	xMsg2501();
	MM2VIS.bMsg2501    := xMsg2501.Q;

	(*  2502 generator DE bearing displacement *)
	xGR_MAX_F_GenBearDE1_Hi(In:= IN_GC.tF_GenBear_DE1.Ai, Gw:= Para.rF_GenBear_Hi, Hy:= 0.0);
	xGR_MAX_F_GenBearDE2_Hi(In:= IN_GC.tF_GenBear_DE2.Ai, Gw:= Para.rF_GenBear_Hi, Hy:= 0.0);

	xMsg2502.Enable    := IN_GC.tPB2MM.bParaSetupOk	AND(Para.bF_GenBear_DE1_Active OR Para.bF_GenBear_DE2_Active);
	xMsg2502.Set       := (xGR_MAX_F_GenBearDE1_Hi.Q AND IN_GC.tF_GenBear_DE1.GoodQual)
					   OR (xGR_MAX_F_GenBearDE2_Hi.Q AND IN_GC.tF_GenBear_DE2.GoodQual);
	xMsg2502.PT        := Para.tiF_GenBear_Hi;
	xMsg2502.RiskClass := 4;
	xMsg2502.Prio      := 4;
	xMsg2502.Reset     := FALSE;
	xMsg2502();
	MM2VIS.bMsg2502    := xMsg2502.Q;

	(*  2503 generator NDE bearing displacement *)
	xGR_MAX_F_GenBearNDE1_Hi(In:= IN_GC.tF_GenBear_NDE1.Ai, Gw:= Para.rF_GenBear_Hi, Hy:= 0.0);
	xGR_MAX_F_GenBearNDE2_Hi(In:= IN_GC.tF_GenBear_NDE2.Ai, Gw:= Para.rF_GenBear_Hi, Hy:= 0.0);

	xMsg2503.Enable    := IN_GC.tPB2MM.bParaSetupOk	AND(Para.bF_GenBear_NDE1_Active OR Para.bF_GenBear_NDE2_Active);
	xMsg2503.Set       := (xGR_MAX_F_GenBearNDE1_Hi.Q AND IN_GC.tF_GenBear_NDE1.GoodQual)
					   OR (xGR_MAX_F_GenBearNDE2_Hi.Q AND IN_GC.tF_GenBear_NDE2.GoodQual);
	xMsg2503.PT        := Para.tiF_GenBear_Hi;
	xMsg2503.RiskClass := 4;
	xMsg2503.Prio      := 4;
	xMsg2503.Reset     := FALSE;
	xMsg2503();
	MM2VIS.bMsg2503    := xMsg2503.Q;

	(* W2504 Generator AVR panel MCB trip *)
	xMsg2504.Enable    := TRUE;
	xMsg2504.Set       := NOT IN_GC.tGenCtr_CktBkr_Trip.Di;
	xMsg2504.PT        := T#0s;
	xMsg2504.RiskClass := 4;
	xMsg2504.Prio      := 4;
	xMsg2504.Reset     := FALSE;
	xMsg2504();
	MM2VIS.bMsg2504    := xMsg2504.Q;

	(* W2505 Oilskid low pressure oil filter clogged *)
	xMsg2505.Enable		:= TRUE;
	xMsg2505.Set		:= bAMM_DPr_OilSkid_FiltLP_Hi;
	xMsg2505.PT			:= T#120s;
	xMsg2505.Prio		:= 4;
	xMsg2505.Reset		:= FALSE;
	xMsg2505();
	MM2VIS.bMsg2505		:= xMsg2505.Q;

	MM2VIS.bMsg2506 ; (*W2506 Oilskid  --> NOT USED *)
	MM2VIS.bMsg2507 ; (*W2507 Oilskid  --> NOT USED *)

	(* W2508 Oilskid high pressure oil filter DE clogged *)
	xMsg2508.Enable		:= TRUE;
	xMsg2508.Set		:= bAMM_DPr_OilSkid_FiltHP_DE_Hi;
	xMsg2508.PT			:= T#10s;
	xMsg2508.Prio		:= 4;
	xMsg2508.Reset		:= FALSE;
	xMsg2508();
	MM2VIS.bMsg2508		:= xMsg2508.Q;

	(* W2555 measuring signal failure generator air inlet temperature *)
	xMsg2555.Enable    := Para.bT_GenAirIn_Active;
	xMsg2555.Set       := IN_GC.tPB2MM.bParaSetupOk AND NOT IN_GC.tGen_T_In.GoodQual;
	xMsg2555.PT        := T#0s;
	xMsg2555.RiskClass := 4;
	xMsg2555.Prio      := 4;
	xMsg2555.Reset     := FALSE;
	xMsg2555();
	MM2VIS.bMsg2555    :=  xMsg2555.Q;

	(* W2556 measuring signal failure generator air outlet temperature *)
	xMsg2556.Enable    := Para.bT_GenAirOut_Active;
	xMsg2556.Set       := IN_GC.tPB2MM.bParaSetupOk AND NOT IN_GC.tT_GenAirOut.GoodQual;
	xMsg2556.PT        := T#0s;
	xMsg2556.RiskClass := 4;
	xMsg2556.Prio      := 4;
	xMsg2556.Reset     := FALSE;
	xMsg2556();
	MM2VIS.bMsg2556    :=  xMsg2556.Q;

	(* W2573 Overvoltage protection generator failure *)
	xMsg2573.Enable    := TRUE;
	xMsg2573.Set       := NOT IN_GC.tU_GenOverVolt.Di;
	xMsg2573.PT        := T#0s;
	xMsg2573.RiskClass := 4;
	xMsg2573.Prio      := 4;
	xMsg2573.Reset     := FALSE;
	xMsg2573();
	MM2VIS.bMsg2573    :=  xMsg2573.Q;

	(*  2631 measuring signal vibration sensor 1 gen.drive end DE bearing *)
	xMsg2631.Enable    := IN_GC.tPB2MM.bParaSetupOk	AND Para.bF_GenBear_DE1_Active;
	xMsg2631.Set       := NOT IN_GC.tF_GenBear_DE1.GoodQual;
	xMsg2631.PT        := T#0s;
	xMsg2631.RiskClass := 4;
	xMsg2631.Prio      := 4;
	xMsg2631.Reset     := FALSE;
	xMsg2631();
	MM2VIS.bMsg2631    :=  xMsg2631.Q;

	(*  2632 measuring signal vibration sensor 2 gen.drive end DE bearing *)
	xMsg2632.Enable    := IN_GC.tPB2MM.bParaSetupOk	AND Para.bF_GenBear_DE2_Active;
	xMsg2632.Set       := NOT IN_GC.tF_GenBear_DE2.GoodQual;
	xMsg2632.PT        := T#0s;
	xMsg2632.RiskClass := 4;
	xMsg2632.Prio      := 4;
	xMsg2632.Reset     := FALSE;
	xMsg2632();
	MM2VIS.bMsg2632    :=  xMsg2632.Q;

	(*  2633 measuring signal vibration sensor 1 gen.non-drive end NDE bearing *)
	xMsg2633.Enable    := IN_GC.tPB2MM.bParaSetupOk	AND Para.bF_GenBear_NDE1_Active;
	xMsg2633.Set       := NOT IN_GC.tF_GenBear_NDE1.GoodQual;
	xMsg2633.PT        := T#0s;
	xMsg2633.RiskClass := 4;
	xMsg2633.Prio      := 4;
	xMsg2633.Reset     := FALSE;
	xMsg2633();
	MM2VIS.bMsg2633    :=  xMsg2633.Q;

	(*  2634 measuring signal vibration sensor 2 gen.non-drive end NDE bearing *)
	xMsg2634.Enable    := IN_GC.tPB2MM.bParaSetupOk	AND Para.bF_GenBear_NDE2_Active;
	xMsg2634.Set       := NOT IN_GC.tF_GenBear_NDE2.GoodQual;
	xMsg2634.PT        := T#0s;
	xMsg2634.RiskClass := 4;
	xMsg2634.Prio      := 4;
	xMsg2634.Reset     := FALSE;
	xMsg2634();
	MM2VIS.bMsg2634    :=  xMsg2634.Q;

	(*  2637 Generator interface panel circuit breaker tripped *)
	xMsg2637.Enable    := TRUE;
	xMsg2637.Set       := NOT IN_GC.tGenIF_CB_On.Di;
	xMsg2637.PT        := T#0s;
	xMsg2637.RiskClass := 4;
	xMsg2637.Prio      := 4;
	xMsg2637.Reset     := FALSE;
	xMsg2637();
	MM2VIS.bMsg2637    :=  xMsg2637.Q;

	(*  2665 Generator heater circuit breaker tripped *)
	xMsg2665.Enable    := TRUE;
	xMsg2665.Set       := NOT IN_GC.tGenHeat_CB_On.Di;
	xMsg2665.PT        := T#0s;
	xMsg2665.RiskClass := 4;
	xMsg2665.Prio      := 4;
	xMsg2665.Reset     := FALSE;
	xMsg2665();
	MM2VIS.bMsg2665    :=  xMsg2665.Q;

	(* W2690 rotor earth fault *)
	xMsg2690.Enable		:= TRUE;
	xMsg2690.Set		:= NOT IN_GC.tGenRotorEarthFault.Di;
	xMsg2690.PT			:= T#0s;
	xMsg2690.Prio		:= 4;
	xMsg2690.RiskClass	:= 4;
	xMsg2690.Reset		:= FALSE;
	xMsg2690();
	MM2VIS.bMsg2690		:= xMsg2690.Q;

	(* W2691 reactive power/undervoltage protection (Q-U-protection) *)
	xMsg2691.Enable		:= TRUE;
	xMsg2691.Set		:= NOT IN_GC.tQ_GenUnderVoltProt.Di;
	xMsg2691.PT			:= T#0s;
	xMsg2691.Prio		:= 4;
	xMsg2691.RiskClass	:= 4;
	xMsg2691.Reset		:= FALSE;
	xMsg2691();
	MM2VIS.bMsg2691		:= xMsg2691.Q;

	(* W3219 excitation voltage low *)
	xMsg3219.Enable    := TRUE;
	xMsg3219.Set       := bU_Gen_Exc_Min AND bU_Gen_Mon_Ena;
	xMsg3219.PT        := T#0s;
	xMsg3219.RiskClass := 4;
	xMsg3219.Prio      := 4;
	xMsg3219.Reset     := FALSE;
	xMsg3219();
	MM2VIS.bMsg3219    := xMsg3219.Q;

	(* A3319 Generator protection trip *)
	xMsg3319.Enable    := TRUE;
	xMsg3319.Set       := NOT IN_GC.tGenPrctTrip.Di AND IN_GC.tGenPrctTrip.GoodQual;
	xMsg3319.PT        := T#0s;
	xMsg3319.RiskClass := 4;
	xMsg3319.Prio      := 2;
	xMsg3319.Reset     := FALSE;
	xMsg3319();
	OUT_GC.bMsg3319    := xMsg3319.Q;
	MM2VIS.bMsg3319    := xMsg3319.Q;

	(* A3393 generator overexcitation *)
	xMsg3393.Enable		:= TRUE;
	xMsg3393.Set		:= NOT IN_GC.tGenOverExc.Di;
	xMsg3393.PT			:= T#0s;
	xMsg3393.Prio		:= 2;
	xMsg3393.RiskClass	:= 4;
	xMsg3393.Reset		:= FALSE;
	xMsg3393();
	MM2VIS.bMsg3393		:= xMsg3393.Q;

	(* W3418 Oilskid oil in oil sump *)
	xMsg3418.Enable		:= TRUE;
	xMsg3418.Set		:= bAMM_Lev_OilSkid_Sump_Hi;
	xMsg3418.PT			:= T#0s;
	xMsg3418.Prio		:= 4;
	xMsg3418.Reset		:= FALSE;
	xMsg3418();
	MM2VIS.bMsg3418		:= xMsg3418.Q;

	(* W3419 Oilskid tank oil level measuring signal failure *)
	xMsg3419.Enable		:= TRUE;
	xMsg3419.Set		:= bAMM_Lev_OilSkid_Tank_Ms;
	xMsg3419.PT			:= T#10s;
	xMsg3419.Prio		:= 4;
	xMsg3419.Reset		:= FALSE;
	xMsg3419();
	MM2VIS.bMsg3419 	:= xMsg3419.Q;

	(* W3420 Oilskid tank oil level low *)
	xMsg3420.Enable		:= TRUE;
	xMsg3420.Set		:= bAMM_Lev_OilSkid_Tank_Lo;
	xMsg3420.PT			:= T#120s;
	xMsg3420.Prio		:= 4;
	xMsg3420.Reset		:= FALSE;
	xMsg3420();
	MM2VIS.bMsg3420		:= xMsg3420.Q;

	(* W3421 Oilskid tank oil temperature measuring signal failure *)
	xMsg3421.Enable		:= TRUE;
	xMsg3421.Set		:= bAMM_T_OilSkid_Tank_Ms;
	xMsg3421.PT			:= T#10s;
	xMsg3421.Prio		:= 4;
	xMsg3421.Reset		:= FALSE;
	xMsg3421();
	MM2VIS.bMsg3421		:= xMsg3421.Q;

	(* W3422 Oilskid tank oil temperature low *)
	xMsg3422.Enable		:= TRUE;
	xMsg3422.Set		:= bAMM_T_OilSkid_Tank_Lo;
	xMsg3422.PT			:= T#0s;
	xMsg3422.Prio		:= 4;
	xMsg3422.Reset		:= FALSE;
	xMsg3422();
	MM2VIS.bMsg3422		:= xMsg3422.Q;

	(* W3423 Oilskid oil supply temperature measuring signal failure *)
	xMsg3423.Enable		:= TRUE;
	xMsg3423.Set		:= bAMM_T_OilSkid_Supply_Ms;
	xMsg3423.PT			:= T#10s;
	xMsg3423.Prio		:= 4;
	xMsg3423.Reset		:= FALSE;
	xMsg3423();
	MM2VIS.bMsg3423		:= xMsg3423.Q;

	(* W3424 Oilskid oil supply temperature low *)
	xMsg3424.Enable		:= TRUE;
	xMsg3424.Set		:= bAMM_T_OilSkid_Supply_Lo;
	xMsg3424.PT			:= T#0s;
	xMsg3424.Prio		:= 4;
	xMsg3424.Reset		:= FALSE;
	xMsg3424();
	MM2VIS.bMsg3424		:= xMsg3424.Q;

	(* W3425 Oilskid oil supply temperature high *)
	xMsg3425.Enable		:= TRUE;
	xMsg3425.Set		:= bAMM_T_OilSkid_Supply_Hi;
	xMsg3425.PT			:= T#0s;
	xMsg3425.Prio		:= 4;
	xMsg3425.Reset		:= FALSE;
	xMsg3425();
	MM2VIS.bMsg3425		:= xMsg3425.Q;

	(* W3426 Oilskid low pressure oil pump circuit breaker tripped *)
	xMsg3426.Enable		:= TRUE;
	xMsg3426.Set		:= bAMM_OilSkid_PumpLP_CB;
	xMsg3426.PT			:= T#0s;
	xMsg3426.Prio		:= 4;
	xMsg3426.Reset		:= FALSE;
	xMsg3426();
	MM2VIS.bMsg3426		:= xMsg3426.Q;

	(* W3427 Oilskid oil flow TO DE bearing measuring signal failure *)
	xMsg3427.Enable		:= TRUE;
	xMsg3427.Set		:= bAMM_Flow_OilSkid_DE_Ms;
	xMsg3427.PT			:= T#10s;
	xMsg3427.Prio		:= 4;
	xMsg3427.Reset		:= FALSE;
	xMsg3427();
	MM2VIS.bMsg3427		:= xMsg3427.Q;

	(* W3428 Oilskid oil flow TO DE bearing low *)
	xMsg3428.Enable		:= TRUE;
	xMsg3428.Set		:= bAMM_Flow_OilSkid_DE_Lo;
	xMsg3428.PT			:= T#120s;
	xMsg3428.Prio		:= 4;
	xMsg3428.Reset		:= FALSE;
	xMsg3428();
	MM2VIS.bMsg3428		:= xMsg3428.Q;

	(* W3429 Oilskid oil flow TO DE bearing high *)
	xMsg3429.Enable		:= TRUE;
	xMsg3429.Set		:= bAMM_Flow_OilSkid_DE_Hi;
	xMsg3429.PT			:= T#120s;
	xMsg3429.Prio		:= 4;
	xMsg3429.Reset		:= FALSE;
	xMsg3429();
	MM2VIS.bMsg3429		:= xMsg3429.Q;

	(* W3430 Oilskid oil flow TO NDE bearing measuring signal failure *)
	xMsg3430.Enable		:= TRUE;
	xMsg3430.Set		:= bAMM_Flow_OilSkid_NDE_Ms;
	xMsg3430.PT			:= T#10s;
	xMsg3430.Prio		:= 4;
	xMsg3430.Reset		:= FALSE;
	xMsg3430();
	MM2VIS.bMsg3430		:= xMsg3430.Q;

	(* W3431 Oilskid oil flow TO NDE bearing low *)
	xMsg3431.Enable		:= TRUE;
	xMsg3431.Set		:= bAMM_Flow_OilSkid_NDE_Lo;
	xMsg3431.PT			:= T#120s;
	xMsg3431.Prio		:= 4;
	xMsg3431.Reset		:= FALSE;
	xMsg3431();
	MM2VIS.bMsg3431		:= xMsg3431.Q;

	(* W3432 Oilskid oil flow TO NDE bearing high *)
	xMsg3432.Enable		:= TRUE;
	xMsg3432.Set		:= bAMM_Flow_OilSkid_NDE_Hi;
	xMsg3432.PT			:= T#120s;
	xMsg3432.Prio		:= 4;
	xMsg3432.Reset		:= FALSE;
	xMsg3432();
	MM2VIS.bMsg3432		:= xMsg3432.Q;

	(* W3433 Oilskid high pressure oil pump circuit breaker tripped *)
	xMsg3433.Enable		:= TRUE;
	xMsg3433.Set		:= bAMM_OilSkid_PumpHP_CB;
	xMsg3433.PT			:= T#0s;
	xMsg3433.Prio		:= 4;
	xMsg3433.Reset		:= FALSE;
	xMsg3433();
	MM2VIS.bMsg3433		:= xMsg3433.Q;

	(* W3434 Oilskid high pressure oil pump circuit breaker tripped - UPS *)
	xMsg3434.Enable		:= TRUE;
	xMsg3434.Set		:= bAMM_OilSkid_PumpHP_CB_UPS;
	xMsg3434.PT			:= T#0s;
	xMsg3434.Prio		:= 4;
	xMsg3434.Reset		:= FALSE;
	xMsg3434();
	MM2VIS.bMsg3434		:= xMsg3434.Q;

	(* W3435 Oilskid oil pressure TO DE bearing measuring signal failure *)
	xMsg3435.Enable		:= TRUE;
	xMsg3435.Set		:= bAMM_Pr_OilSkid_HP_DE_Ms;
	xMsg3435.PT			:= T#10s;
	xMsg3435.Prio		:= 4;
	xMsg3435.Reset		:= FALSE;
	xMsg3435();
	MM2VIS.bMsg3435		:= xMsg3435.Q;

	(* W3436 Oilskid oil pressure TO DE bearing low *)
	xMsg3436.Enable		:= TRUE;
	xMsg3436.Set		:= bAMM_Pr_OilSkid_HP_DE_Lo;
	xMsg3436.PT			:= T#0s;
	xMsg3436.Prio		:= 4;
	xMsg3436.Reset		:= FALSE;
	xMsg3436();
	MM2VIS.bMsg3436		:= xMsg3436.Q;

	(* W3437 Oilskid fan circuit breaker tripped*)
	xMsg3437.Enable		:= TRUE;
	xMsg3437.Set		:= bAMM_OilSkid_Fan_CB;
	xMsg3437.PT			:= T#0s;
	xMsg3437.Prio		:= 4;
	xMsg3437.Reset		:= FALSE;
	xMsg3437();
	MM2VIS.bMsg3437		:= xMsg3437.Q;

	(* W3438 Oilskid heater circuit breaker tripped *)
	xMsg3438.Enable		:= TRUE;
	xMsg3438.Set		:= bAMM_OilSkid_Heater_CB;
	xMsg3438.PT			:= T#0s;
	xMsg3438.Prio		:= 4;
	xMsg3438.Reset		:= FALSE;
	xMsg3438();
	MM2VIS.bMsg3438		:= xMsg3438.Q;

	(* W3439 Oilskid main switch auxiliaries opened *)
	xMsg3439.Enable		:= TRUE;
	xMsg3439.Set		:= bAMM_OilSkid_MCB;
	xMsg3439.PT			:= T#0s;
	xMsg3439.Prio		:= 4;
	xMsg3439.Reset		:= FALSE;
	xMsg3439();
	MM2VIS.bMsg3439		:= xMsg3439.Q;

	(* W3440 Oilskid auxiliaries voltage NOT available *)
	xMsg3440.Enable		:= TRUE;
	xMsg3440.Set		:= bAMM_OilSkid_AuxV;
	xMsg3440.PT			:= T#2s;
	xMsg3440.Prio		:= 4;
	xMsg3440.Reset		:= FALSE;
	xMsg3440();
	MM2VIS.bMsg3440		:= xMsg3440.Q;

	(* W3441 Oilskid auxiliaries voltage NOT available - UPS *)
	xMsg3441.Enable		:= TRUE;
	xMsg3441.Set		:= bAMM_OilSkid_AuxV_UPS;
	xMsg3441.PT			:= T#0s;
	xMsg3441.Prio		:= 4;
	xMsg3441.Reset		:= FALSE;
	xMsg3441();
	MM2VIS.bMsg3441		:= xMsg3441.Q;

	(* W3442 Oilskid oil pressure TO NDE bearing measuring signal failure *)
	xMsg3442.Enable		:= TRUE;
	xMsg3442.Set		:= bAMM_Pr_OilSkid_HP_NDE_Ms;
	xMsg3442.PT			:= T#10s;
	xMsg3442.Prio		:= 4;
	xMsg3442.Reset		:= FALSE;
	xMsg3442();
	MM2VIS.bMsg3442		:= xMsg3442.Q;

	(* W3443 Oilskid oil pressure TO NDE bearing low *)
	xMsg3443.Enable		:= TRUE;
	xMsg3443.Set		:= bAMM_Pr_OilSkid_HP_NDE_Lo;
	xMsg3443.PT			:= T#0s;
	xMsg3443.Prio		:= 4;
	xMsg3443.Reset		:= FALSE;
	xMsg3443();
	MM2VIS.bMsg3443		:= xMsg3443.Q;

	(* W3446 Oilskid high pressure oil filter NDE clogged *)
	xMsg3446.Enable		:= TRUE;
	xMsg3446.Set		:= bAMM_DPr_OilSkid_FiltHP_NDE_Hi;
	xMsg3446.PT			:= T#10s;
	xMsg3446.Prio		:= 4;
	xMsg3446.Reset		:= FALSE;
	xMsg3446();
	MM2VIS.bMsg3446		:= xMsg3446.Q;

	(* W3447 Oilskid circulation pump circuit breaker tripped *)
	xMsg3447.Enable		:= TRUE;
	xMsg3447.Set		:= bAMM_OilSkid_PumpC_CB;
	xMsg3447.PT			:= T#0s;
	xMsg3447.Prio		:= 4;
	xMsg3447.Reset		:= FALSE;
	xMsg3447();
	MM2VIS.bMsg3447		:= xMsg3447.Q;

	(* W3468 generator air inlet temperature 2 signal failure *)
	xMsg3468.Enable		:= Para.bT_GenAirIn2_Active;
	xMsg3468.Set		:= IN_GC.tPB2MM.bParaSetupOk AND NOT IN_GC.tGen_T_In2.GoodQual;
	xMsg3468.PT			:= T#0s;
	xMsg3468.Prio		:= 4;
	xMsg3468.Reset		:= FALSE;
	xMsg3468();
	MM2VIS.bMsg3468		:= xMsg3468.Q;

	(* W3516 Excitation voltage high *)
	xMsg3516.Enable    := TRUE;
	xMsg3516.Set       := bU_Gen_Exc_Max AND IN_GC.tEng_Run.Do;
	xMsg3516.PT        := T#0s;
	xMsg3516.RiskClass := 4;
	xMsg3516.Prio      := 4;
	xMsg3516.Reset     := FALSE;
	xMsg3516();
	MM2VIS.bMsg3516    := xMsg3516.Q;

	(* W3563 Generator lubrication failure *)
	xMsg3563.Enable    := TRUE;
	xMsg3563.Set       := IN_GC.bIgn_Dem AND NOT IN_GC.tFlow_Gen_Lube.Di;
	xMsg3563.PT        := T#5s;
	xMsg3563.RiskClass := 4;
	xMsg3563.Prio      := 4;
	xMsg3563.Reset     := FALSE;
	xMsg3563();
	MM2VIS.bMsg3563    :=  xMsg3563.Q;

	(* W3566 Messignalstörung Generator Leistungsfaktorsollwert *)
	xMsg3566.Enable    := FALSE;(*->3593*)
	xMsg3566.Set       := FALSE;
	xMsg3566.PT        := T#0s;
	xMsg3566.Prio      := 4;
	xMsg3566.Reset     := FALSE;
	xMsg3566();
	MM2VIS.bMsg3566    := xMsg3566.Q;

	(* W3573 Failure Generator lubricating oil - Cooling *)(* A2336 *)
	xMsg3573.Enable    := FALSE;
	xMsg3573.Set       := NOT IN_GC.tGen_LO_CoolingSys_Fail.Di;
	xMsg3573.PT        := T#0s;
	xMsg3573.RiskClass := 4;
	xMsg3573.Prio      := 4;
	xMsg3573.Reset     := FALSE;
	xMsg3573();
	MM2VIS.bMsg3573    := xMsg3573.Q;

	(* W9311 Earth failure generator *)(* A1134 *)
	xMsg9311.Enable    := TRUE;
	xMsg9311.Set       := NOT IN_GC.tGndFaultW.Di;
	xMsg9311.PT        := T#0s;
	xMsg9311.RiskClass := 4;
	xMsg9311.Prio      := 4;
	xMsg9311.Reset     := FALSE;
	xMsg9311();
	MM2VIS.bMsg9311    := xMsg9311.Q;

	(* counter Earth fault with running engine *)
	xTON_SecTick(IN:= NOT xTON_SecTick.Q, PT:= T#800ms);(*800ms! = 1s tick*)

	IF ((NOT IN_GC.tGndFaultW.Di) OR bMsg9372_set) AND IN_GC.tEng_Run.Do AND xTON_SecTick.Q AND IN_GC.tPB2MM.bParaSetupOk THEN
		iOpS_GndFailure	:= iOpS_GndFailure + 1;
	END_IF;

	IF iOpS_GndFailure >= 60 THEN
		iOpS_GndFailure	:= 0;
		iOpM_GndFailure	:= iOpM_GndFailure + 1;
	END_IF;

	IF iOpM_GndFailure >= 60 THEN
		iOpM_GndFailure	:= 0;
		VIS2MM.iOpH_GndFailure := VIS2MM.iOpH_GndFailure + 1;
	END_IF;

	(* check limits *)
	IF VIS2MM.iOpH_GndFailure >= 1000000000 THEN
		VIS2MM.iOpH_GndFailure := VIS2MM.iOpH_GndFailure - 1000000000;		(* check upper limit *)
	ELSIF VIS2MM.iOpH_GndFailure <= -1000000000 THEN
		VIS2MM.iOpH_GndFailure := VIS2MM.iOpH_GndFailure + 1000000000;		(* check lower limit *)
	END_IF;

	(* W9285 Measuring signal failure external voltage setpoint *)
	xMsg9285.Enable := 	IN_GC.tU_SetExtAI_Norm.Exist AND IN_GC.tPB2MM.bParaSetupOk;
	xMsg9285.Set := 	bMsg9285;
	xMsg9285.PT := 		T#1s;
	xMsg9285.Prio := 	4;
	xMsg9285.Reset := 	FALSE;
	xMsg9285();
	OUT_GC.bMsg9285 :=	xMsg9285.Q;

	(* W9351 Measuring signal failure external reactive power set point for voltage droop mode *)
	xMsg9351.Enable := 	IN_GC.tQ_Droop_Set.Exist AND IN_GC.tPB2MM.bParaSetupOk;
	xMsg9351.Set := 	bMsg9351;
	xMsg9351.PT := 		T#1s;
	xMsg9351.Prio := 	4;
	xMsg9351.Reset := 	FALSE;
	xMsg9351();
	MM2VIS.bMsg9351    := xMsg9351.Q;

	(* W9365 Automatic generator greasing system error (drive end DE bearing) *)
	xMsg9365.Enable	:= 	TRUE;
	xMsg9365.Set 	:=	IN_GC.bEng_Dem AND IN_GC.tEng_Run.Do AND NOT IN_GC.tGenBearGreasSys2DE.Di;
	xMsg9365.PT 	:=	T#5s;
	xMsg9365.Prio	:= 	4;
	xMsg9365.Reset	:= 	FALSE;
	xMsg9365();
	MM2VIS.bMsg9365	:= xMsg9365.Q;

	(* W9366 Automatic generator greasing system error (non-drive end NDE bearing) *)
	xMsg9366.Enable	:= 	TRUE;
	xMsg9366.Set 	:=	IN_GC.bEng_Dem AND IN_GC.tEng_Run.Do AND NOT IN_GC.tGenBearGreasSys2NDE.Di;
	xMsg9366.PT 	:=	T#5s;
	xMsg9366.Prio	:= 	4;
	xMsg9366.Reset	:= 	FALSE;
	xMsg9366();
	MM2VIS.bMsg9366	:= xMsg9366.Q;

	(* W9367 Automatic generator greasing system - lubrication cartridge empty (drive end DE bearing) *)
	xMsg9367.Enable	:= 	TRUE;
	xMsg9367.Set 	:=	IN_GC.tGenBearGreasSys2DE.Di AND IN_GC.tGenBearGreasSys4DE.Di;
	xMsg9367.PT 	:=	T#5s;
	xMsg9367.Prio	:= 	4;
	xMsg9367.Reset	:= 	FALSE;
	xMsg9367();
	MM2VIS.bMsg9367	:= xMsg9367.Q;

	(* W9368 Automatic generator greasing system - lubrication cartridge empty (non-drive end NDE bearing) *)
	xMsg9368.Enable	:= 	TRUE;
	xMsg9368.Set 	:=	IN_GC.tGenBearGreasSys2NDE.Di AND IN_GC.tGenBearGreasSys4NDE.Di;
	xMsg9368.PT 	:=	T#5s;
	xMsg9368.Prio	:= 	4;
	xMsg9368.Reset	:= 	FALSE;
	xMsg9368();
	MM2VIS.bMsg9368	:= xMsg9368.Q;

	(* W9372 Earth failure generator (MMD) *)
	xMsg9372.Enable	:= 	NOT IN_GC.bSimWinMOD_Active;
	xMsg9372.Set 	:=	bMsg9372_set;
	xMsg9372.PT 	:=	T#0s;
	xMsg9372.Prio	:= 	4;
	xMsg9372.Reset	:= 	FALSE;
	xMsg9372();
	MM2VIS.bMsg9372	:= xMsg9372.Q;

	(*---------------------------------------------------------------------------*)
	(* Operating messages *)

	(* B2156 Q reduction by gen.winding temp. (diagn.msg RPS) *)
	xTP_Msg2156(IN:= bMsg2156, PT := T#60s);

 	xMsg2156.Enable    := TRUE;
	xMsg2156.Set       := xTP_Msg2156.Q;
	xMsg2156.Reset     := TRUE;
	xMsg2156();
	MM2VIS.bMsg2156    := xMsg2156.Q;

	(* B2157 Q reduction by polradwinkel (diagn.msg RPS) *)
	xTP_Msg2157(IN:= bMsg2157, PT := T#60s);

	xMsg2157.Enable    := TRUE;
	xMsg2157.Set       := xTP_Msg2157.Q;
	xMsg2157.Reset     := TRUE;
	xMsg2157();
	MM2VIS.bMsg2157    := xMsg2157.Q;

	(* B2827 Generator Lube Oil System/ Jacket Oil system ready for start and operation *)	(* --> NOT USED *)
	xMsg2827.Enable		:=	FALSE;
	xMsg2827.Set		:=	FALSE;
	xMsg2827.Reset		:=	TRUE;
	xMsg2827();
	MM2VIS.bMsg2827		:=	xMsg2827.Q;

	(* B2828 Generator Lube Oil System - Oil outlet pressure ok *)							(* --> NOT USED *)
	xMsg2828.Enable		:=	FALSE;
	xMsg2828.Set		:=	FALSE;
	xMsg2828.Reset		:=	TRUE;
	xMsg2828();
	MM2VIS.bMsg2828		:=	xMsg2828.Q;

	(* B2829 Generator Lube Oil System - drive end bearing oil flow ok*)					(* --> NOT USED *)
	xMsg2829.Enable		:=	FALSE;
	xMsg2829.Set		:=	FALSE;
	xMsg2829.Reset		:=	TRUE;
	xMsg2829();
	MM2VIS.bMsg2829		:=	xMsg2829.Q;

	(* B2830 Generator Lube Oil System - non drive end bearing oil flow ok*)				(* --> NOT USED *)
	xMsg2830.Enable		:=	FALSE;
	xMsg2830.Set		:=	FALSE;
	xMsg2830.Reset		:=	TRUE;
	xMsg2830();
	MM2VIS.bMsg2830		:=	xMsg2830.Q;

	(* B2998 reactive power limitation by under voltage *)
	xTP_Msg2998(IN:= bMsg2998, PT := T#60s);

	xMsg2998.Enable		:=	TRUE;
	xMsg2998.Set		:=	xTP_Msg2998.Q;
	xMsg2998.Reset		:=	TRUE;
	xMsg2998();
	MM2VIS.bMsg2998		:=	xMsg2998.Q;

	(* B template
	xMsg.Enable		:=	TRUE;
	xMsg.Set		:=	bBool;
	xMsg.Reset		:=	TRUE;
	xMsg();
	MM2VIS.bMsg		:=	xMsg.Q;	*)

	(*---------------------------------------------------------------------------*)
	(* general alarms for further module operations *)
	bGnlTrip1   := OUT_GC.tGC2AB.bGnlTrip1   OR IN_GC.tAB2GC.bGnlTrip1;
	bGnlTrip2   := OUT_GC.tGC2AB.bGnlTrip2   OR IN_GC.tAB2GC.bGnlTrip2;
	bGnlTrip3   := OUT_GC.tGC2AB.bGnlTrip3   OR IN_GC.tAB2GC.bGnlTrip3;
	bGnlWarning := OUT_GC.tGC2AB.bGnlWarning OR IN_GC.tAB2GC.bGnlWarning;

	bGnlTrip	:= bGnlTrip1 OR bGnlTrip2 OR bGnlTrip3;

	(*******************************************************************************)

END_PROGRAM
```

#### MsgGCInit.st
```iecst
(*******************************************************************************
Msg_VE	 			 alarms generation MM_ventilation

This code is confidential and proprietary to the INNIO Company.
It may not be used in any form, or reproduced in any manner,
without written permission of the INNIO Company.
Copyright, INNIO Company, 2019

Customized modifications: -
------------------------

History:
-------
V0.00.0	29.07.2011	lettenb.	new

Instructions for use:
--------------------
1) declare alarm with function block "Msg"

2) use template to create a new alarm, substitue 0000 by message number:

	xMsg0000.Num		:=	0000;					alarm number
	xMsg0000.AmmSysAdr	:=  iAdrAmmBase2MM;			do not change
	xMsg0000.AmmOutAdr	:=  iAdrMM2AmmBase;			do not change

3) 	set alarm number

Outstandings:
------------
(*******************************************************************************)
PROGRAM _INIT

	iAdrAmmBase2MM		:=  ADR(IN_GC.tAB2GC);
	iAdrMM2AmmBase		:=  ADR(OUT_GC.tGC2AB);

	(*---------------------------------------------------------------------------*)
	xMsg1036.Num       := 1036;
	xMsg1036.AmmInAdr  := iAdrAmmBase2MM;
	xMsg1036.AmmOutAdr := iAdrMM2AmmBase;

	xMsg1037.Num       := 1037;
	xMsg1037.AmmInAdr  := iAdrAmmBase2MM;
	xMsg1037.AmmOutAdr := iAdrMM2AmmBase;

	xMsg1038.Num       := 1038;
	xMsg1038.AmmInAdr  := iAdrAmmBase2MM;
	xMsg1038.AmmOutAdr := iAdrMM2AmmBase;

	xMsg1062.Num       := 1062;
	xMsg1062.AmmInAdr  := iAdrAmmBase2MM;
	xMsg1062.AmmOutAdr := iAdrMM2AmmBase;

	xMsg1073.Num       := 1073;
	xMsg1073.AmmInAdr  := iAdrAmmBase2MM;
	xMsg1073.AmmOutAdr := iAdrMM2AmmBase;

	xMsg1109.Num       := 1109;
	xMsg1109.AmmInAdr  := iAdrAmmBase2MM;
	xMsg1109.AmmOutAdr := iAdrMM2AmmBase;

	xMsg1110.Num       := 1110;
	xMsg1110.AmmInAdr  := iAdrAmmBase2MM;
	xMsg1110.AmmOutAdr := iAdrMM2AmmBase;

	xMsg1111.Num       := 1111;
	xMsg1111.AmmInAdr  := iAdrAmmBase2MM;
	xMsg1111.AmmOutAdr := iAdrMM2AmmBase;

	xMsg1112.Num       := 1112;
	xMsg1112.AmmInAdr  := iAdrAmmBase2MM;
	xMsg1112.AmmOutAdr := iAdrMM2AmmBase;

	xMsg1113.Num       := 1113;
	xMsg1113.AmmInAdr  := iAdrAmmBase2MM;
	xMsg1113.AmmOutAdr := iAdrMM2AmmBase;

	xMsg1121.Num       := 1121;
	xMsg1121.AmmInAdr  := iAdrAmmBase2MM;
	xMsg1121.AmmOutAdr := iAdrMM2AmmBase;

	xMsg1122.Num       := 1122;
	xMsg1122.AmmInAdr  := iAdrAmmBase2MM;
	xMsg1122.AmmOutAdr := iAdrMM2AmmBase;

	xMsg1123.Num       := 1123;
	xMsg1123.AmmInAdr  := iAdrAmmBase2MM;
	xMsg1123.AmmOutAdr := iAdrMM2AmmBase;

	xMsg1124.Num       := 1124;
	xMsg1124.AmmInAdr  := iAdrAmmBase2MM;
	xMsg1124.AmmOutAdr := iAdrMM2AmmBase;

	xMsg1125.Num       := 1125;
	xMsg1125.AmmInAdr  := iAdrAmmBase2MM;
	xMsg1125.AmmOutAdr := iAdrMM2AmmBase;

	xMsg1126.Num       := 1126;
	xMsg1126.AmmInAdr  := iAdrAmmBase2MM;
	xMsg1126.AmmOutAdr := iAdrMM2AmmBase;

	xMsg1127.Num       := 1127;
	xMsg1127.AmmInAdr  := iAdrAmmBase2MM;
	xMsg1127.AmmOutAdr := iAdrMM2AmmBase;

	xMsg1132.Num       := 1132;
	xMsg1132.AmmInAdr  := iAdrAmmBase2MM;
	xMsg1132.AmmOutAdr := iAdrMM2AmmBase;

	xMsg1134.Num       := 1134;
	xMsg1134.AmmInAdr  := iAdrAmmBase2MM;
	xMsg1134.AmmOutAdr := iAdrMM2AmmBase;

	xMsg1143.Num       := 1143;
	xMsg1143.AmmInAdr  := iAdrAmmBase2MM;
	xMsg1143.AmmOutAdr := iAdrMM2AmmBase;

	xMsg1144.Num       := 1144;
	xMsg1144.AmmInAdr  := iAdrAmmBase2MM;
	xMsg1144.AmmOutAdr := iAdrMM2AmmBase;

	xMsg1154.Num       := 1154;
	xMsg1154.AmmInAdr  := iAdrAmmBase2MM;
	xMsg1154.AmmOutAdr := iAdrMM2AmmBase;

	xMsg1155.Num       := 1155;
	xMsg1155.AmmInAdr  := iAdrAmmBase2MM;
	xMsg1155.AmmOutAdr := iAdrMM2AmmBase;

	xMsg1156.Num       := 1156;
	xMsg1156.AmmInAdr  := iAdrAmmBase2MM;
	xMsg1156.AmmOutAdr := iAdrMM2AmmBase;

	xMsg1157.Num       := 1157;
	xMsg1157.AmmInAdr  := iAdrAmmBase2MM;
	xMsg1157.AmmOutAdr := iAdrMM2AmmBase;

	xMsg1158.Num       := 1158;
	xMsg1158.AmmInAdr  := iAdrAmmBase2MM;
	xMsg1158.AmmOutAdr := iAdrMM2AmmBase;

	xMsg1185.Num       := 1185;
	xMsg1185.AmmInAdr  := iAdrAmmBase2MM;
	xMsg1185.AmmOutAdr := iAdrMM2AmmBase;

	xMsg2100.Num       := 2100;
	xMsg2100.AmmInAdr  := iAdrAmmBase2MM;
	xMsg2100.AmmOutAdr := iAdrMM2AmmBase;

	xMsg2105.Num       := 2105;
	xMsg2105.AmmInAdr  := iAdrAmmBase2MM;
	xMsg2105.AmmOutAdr := iAdrMM2AmmBase;

	xMsg2106.Num       := 2106;
	xMsg2106.AmmInAdr  := iAdrAmmBase2MM;
	xMsg2106.AmmOutAdr := iAdrMM2AmmBase;

	xMsg2107.Num       := 2107;
	xMsg2107.AmmInAdr  := iAdrAmmBase2MM;
	xMsg2107.AmmOutAdr := iAdrMM2AmmBase;

	xMsg2108.Num       := 2108;
	xMsg2108.AmmInAdr  := iAdrAmmBase2MM;
	xMsg2108.AmmOutAdr := iAdrMM2AmmBase;

	xMsg2109.Num       := 2109;
	xMsg2109.AmmInAdr  := iAdrAmmBase2MM;
	xMsg2109.AmmOutAdr := iAdrMM2AmmBase;

	xMsg2110.Num       := 2110;
	xMsg2110.AmmInAdr  := iAdrAmmBase2MM;
	xMsg2110.AmmOutAdr := iAdrMM2AmmBase;

	xMsg2115.Num       := 2115;
	xMsg2115.AmmInAdr  := iAdrAmmBase2MM;
	xMsg2115.AmmOutAdr := iAdrMM2AmmBase;

	xMsg2156.Num       := 2156;
	xMsg2156.AmmInAdr  := iAdrAmmBase2MM;
	xMsg2156.AmmOutAdr := iAdrMM2AmmBase;

	xMsg2157.Num       := 2157;
	xMsg2157.AmmInAdr  := iAdrAmmBase2MM;
	xMsg2157.AmmOutAdr := iAdrMM2AmmBase;

	xMsg2202.Num       := 2202;
	xMsg2202.AmmInAdr  := iAdrAmmBase2MM;
	xMsg2202.AmmOutAdr := iAdrMM2AmmBase;

	xMsg2203.Num       := 2203;
	xMsg2203.AmmInAdr  := iAdrAmmBase2MM;
	xMsg2203.AmmOutAdr := iAdrMM2AmmBase;

	xMsg2204.Num       := 2204;
	xMsg2204.AmmInAdr  := iAdrAmmBase2MM;
	xMsg2204.AmmOutAdr := iAdrMM2AmmBase;

	xMsg2205.Num       := 2205;
	xMsg2205.AmmInAdr  := iAdrAmmBase2MM;
	xMsg2205.AmmOutAdr := iAdrMM2AmmBase;

	xMsg2206.Num       := 2206;
	xMsg2206.AmmInAdr  := iAdrAmmBase2MM;
	xMsg2206.AmmOutAdr := iAdrMM2AmmBase;

	xMsg2207.Num       := 2207;
	xMsg2207.AmmInAdr  := iAdrAmmBase2MM;
	xMsg2207.AmmOutAdr := iAdrMM2AmmBase;

	xMsg2208.Num 	   := 2208;
	xMsg2208.AmmInAdr  := iAdrAmmBase2MM;
	xMsg2208.AmmOutAdr := iAdrMM2AmmBase;

	xMsg2277.Num       := 2277;
	xMsg2277.AmmInAdr  := iAdrAmmBase2MM;
	xMsg2277.AmmOutAdr := iAdrMM2AmmBase;

	xMsg2316.Num       := 2316;
	xMsg2316.AmmInAdr  := iAdrAmmBase2MM;
	xMsg2316.AmmOutAdr := iAdrMM2AmmBase;

	xMsg2336.Num       := 2336;
	xMsg2336.AmmInAdr  := iAdrAmmBase2MM;
	xMsg2336.AmmOutAdr := iAdrMM2AmmBase;

	xMsg2371.Num	   := 2371;
	xMsg2371.AmmInAdr  := iAdrAmmBase2MM;
	xMsg2371.AmmOutAdr := iAdrMM2AmmBase;

	xMsg2372.Num	   := 2372;
	xMsg2372.AmmInAdr  := iAdrAmmBase2MM;
	xMsg2372.AmmOutAdr := iAdrMM2AmmBase;

	xMsg2373.Num	   := 2373;
	xMsg2373.AmmInAdr  := iAdrAmmBase2MM;
	xMsg2373.AmmOutAdr := iAdrMM2AmmBase;

	xMsg2501.Num       := 2501;
	xMsg2501.AmmInAdr  := iAdrAmmBase2MM;
	xMsg2501.AmmOutAdr := iAdrMM2AmmBase;

	xMsg2502.Num       := 2502;
	xMsg2502.AmmInAdr  := iAdrAmmBase2MM;
	xMsg2502.AmmOutAdr := iAdrMM2AmmBase;

	xMsg2503.Num       := 2503;
	xMsg2503.AmmInAdr  := iAdrAmmBase2MM;
	xMsg2503.AmmOutAdr := iAdrMM2AmmBase;

	xMsg2504.Num       := 2504;
	xMsg2504.AmmInAdr  := iAdrAmmBase2MM;
	xMsg2504.AmmOutAdr := iAdrMM2AmmBase;

	xMsg2505.Num 	   := 2505;
	xMsg2505.AmmInAdr  := iAdrAmmBase2MM;
	xMsg2505.AmmOutAdr := iAdrMM2AmmBase;

	xMsg2508.Num 	   := 2508;
	xMsg2508.AmmInAdr  := iAdrAmmBase2MM;
	xMsg2508.AmmOutAdr := iAdrMM2AmmBase;

	xMsg2555.Num       := 2555;
	xMsg2555.AmmInAdr  := iAdrAmmBase2MM;
	xMsg2555.AmmOutAdr := iAdrMM2AmmBase;

	xMsg2556.Num       := 2556;
	xMsg2556.AmmInAdr  := iAdrAmmBase2MM;
	xMsg2556.AmmOutAdr := iAdrMM2AmmBase;

	xMsg2573.Num       := 2573;
	xMsg2573.AmmInAdr  := iAdrAmmBase2MM;
	xMsg2573.AmmOutAdr := iAdrMM2AmmBase;

	xMsg2631.Num       := 2631;
	xMsg2631.AmmInAdr  := iAdrAmmBase2MM;
	xMsg2631.AmmOutAdr := iAdrMM2AmmBase;

	xMsg2632.Num       := 2632;
	xMsg2632.AmmInAdr  := iAdrAmmBase2MM;
	xMsg2632.AmmOutAdr := iAdrMM2AmmBase;

	xMsg2633.Num       := 2633;
	xMsg2633.AmmInAdr  := iAdrAmmBase2MM;
	xMsg2633.AmmOutAdr := iAdrMM2AmmBase;

	xMsg2634.Num       := 2634;
	xMsg2634.AmmInAdr  := iAdrAmmBase2MM;
	xMsg2634.AmmOutAdr := iAdrMM2AmmBase;

	xMsg2637.Num       := 2637;
	xMsg2637.AmmInAdr  := iAdrAmmBase2MM;
	xMsg2637.AmmOutAdr := iAdrMM2AmmBase;

	xMsg2665.Num       := 2665;
	xMsg2665.AmmInAdr  := iAdrAmmBase2MM;
	xMsg2665.AmmOutAdr := iAdrMM2AmmBase;

	xMsg2690.Num		:=	2690;
	xMsg2690.AmmInAdr	:=  iAdrAmmBase2MM;
	xMsg2690.AmmOutAdr	:=  iAdrMM2AmmBase;

	xMsg2691.Num		:=	2691;
	xMsg2691.AmmInAdr	:=  iAdrAmmBase2MM;
	xMsg2691.AmmOutAdr	:=  iAdrMM2AmmBase;

	xMsg2827.Num	   := 2827;
	xMsg2827.AmmInAdr  := iAdrAmmBase2MM;
	xMsg2827.AmmOutAdr := iAdrMM2AmmBase;

	xMsg2828.Num	   := 2828;
	xMsg2828.AmmInAdr  := iAdrAmmBase2MM;
	xMsg2828.AmmOutAdr := iAdrMM2AmmBase;

	xMsg2829.Num	   := 2829;
	xMsg2829.AmmInAdr  := iAdrAmmBase2MM;
	xMsg2829.AmmOutAdr := iAdrMM2AmmBase;

	xMsg2830.Num	   := 2830;
	xMsg2830.AmmInAdr  := iAdrAmmBase2MM;
	xMsg2830.AmmOutAdr := iAdrMM2AmmBase;

	xMsg2998.Num	   := 2998;
	xMsg2998.AmmInAdr  := iAdrAmmBase2MM;
	xMsg2998.AmmOutAdr := iAdrMM2AmmBase;

	xMsg3219.Num       := 3219;
	xMsg3219.AmmInAdr  := iAdrAmmBase2MM;
	xMsg3219.AmmOutAdr := iAdrMM2AmmBase;

	xMsg3298.Num       := 3298;
	xMsg3298.AmmInAdr  := iAdrAmmBase2MM;
	xMsg3298.AmmOutAdr := iAdrMM2AmmBase;

	xMsg3299.Num       := 3299;
	xMsg3299.AmmInAdr  := iAdrAmmBase2MM;
	xMsg3299.AmmOutAdr := iAdrMM2AmmBase;

	xMsg3319.Num       := 3319;
	xMsg3319.AmmInAdr  := iAdrAmmBase2MM;
	xMsg3319.AmmOutAdr := iAdrMM2AmmBase;

	xMsg3393.Num		:=  3393;
	xMsg3393.AmmInAdr	:=  iAdrAmmBase2MM;
	xMsg3393.AmmOutAdr	:=  iAdrMM2AmmBase;

	xMsg3418.Num 		:= 3418;
	xMsg3418.AmmInAdr 	:= iAdrAmmBase2MM;
	xMsg3418.AmmOutAdr 	:= iAdrMM2AmmBase;

	xMsg3419.Num 		:= 3419;
	xMsg3419.AmmInAdr 	:= iAdrAmmBase2MM;
	xMsg3419.AmmOutAdr 	:= iAdrMM2AmmBase;

	xMsg3420.Num 		:= 3420;
	xMsg3420.AmmInAdr 	:= iAdrAmmBase2MM;
	xMsg3420.AmmOutAdr 	:= iAdrMM2AmmBase;

	xMsg3421.Num 		:= 3421;
	xMsg3421.AmmInAdr 	:= iAdrAmmBase2MM;
	xMsg3421.AmmOutAdr 	:= iAdrMM2AmmBase;

	xMsg3422.Num 		:= 3422;
	xMsg3422.AmmInAdr 	:= iAdrAmmBase2MM;
	xMsg3422.AmmOutAdr 	:= iAdrMM2AmmBase;

	xMsg3423.Num 		:= 3423;
	xMsg3423.AmmInAdr 	:= iAdrAmmBase2MM;
	xMsg3423.AmmOutAdr 	:= iAdrMM2AmmBase;

	xMsg3424.Num 		:= 3424;
	xMsg3424.AmmInAdr 	:= iAdrAmmBase2MM;
	xMsg3424.AmmOutAdr 	:= iAdrMM2AmmBase;

	xMsg3425.Num 		:= 3425;
	xMsg3425.AmmInAdr 	:= iAdrAmmBase2MM;
	xMsg3425.AmmOutAdr 	:= iAdrMM2AmmBase;

	xMsg3426.Num 		:= 3426;
	xMsg3426.AmmInAdr 	:= iAdrAmmBase2MM;
	xMsg3426.AmmOutAdr 	:= iAdrMM2AmmBase;

	xMsg3427.Num 		:= 3427;
	xMsg3427.AmmInAdr 	:= iAdrAmmBase2MM;
	xMsg3427.AmmOutAdr 	:= iAdrMM2AmmBase;

	xMsg3428.Num 		:= 3428;
	xMsg3428.AmmInAdr 	:= iAdrAmmBase2MM;
	xMsg3428.AmmOutAdr 	:= iAdrMM2AmmBase;

	xMsg3429.Num 		:= 3429;
	xMsg3429.AmmInAdr 	:= iAdrAmmBase2MM;
	xMsg3429.AmmOutAdr 	:= iAdrMM2AmmBase;

	xMsg3430.Num 		:= 3430;
	xMsg3430.AmmInAdr 	:= iAdrAmmBase2MM;
	xMsg3430.AmmOutAdr 	:= iAdrMM2AmmBase;

	xMsg3431.Num 		:= 3431;
	xMsg3431.AmmInAdr 	:= iAdrAmmBase2MM;
	xMsg3431.AmmOutAdr 	:= iAdrMM2AmmBase;

	xMsg3432.Num 		:= 3432;
	xMsg3432.AmmInAdr 	:= iAdrAmmBase2MM;
	xMsg3432.AmmOutAdr 	:= iAdrMM2AmmBase;

	xMsg3433.Num 		:= 3433;
	xMsg3433.AmmInAdr 	:= iAdrAmmBase2MM;
	xMsg3433.AmmOutAdr 	:= iAdrMM2AmmBase;

	xMsg3434.Num 		:= 3434;
	xMsg3434.AmmInAdr 	:= iAdrAmmBase2MM;
	xMsg3434.AmmOutAdr 	:= iAdrMM2AmmBase;

	xMsg3435.Num 		:= 3435;
	xMsg3435.AmmInAdr 	:= iAdrAmmBase2MM;
	xMsg3435.AmmOutAdr 	:= iAdrMM2AmmBase;

	xMsg3436.Num 		:= 3436;
	xMsg3436.AmmInAdr 	:= iAdrAmmBase2MM;
	xMsg3436.AmmOutAdr 	:= iAdrMM2AmmBase;

	xMsg3437.Num 		:= 3437;
	xMsg3437.AmmInAdr 	:= iAdrAmmBase2MM;
	xMsg3437.AmmOutAdr 	:= iAdrMM2AmmBase;

	xMsg3438.Num 		:= 3438;
	xMsg3438.AmmInAdr 	:= iAdrAmmBase2MM;
	xMsg3438.AmmOutAdr 	:= iAdrMM2AmmBase;

	xMsg3439.Num 		:= 3439;
	xMsg3439.AmmInAdr 	:= iAdrAmmBase2MM;
	xMsg3439.AmmOutAdr 	:= iAdrMM2AmmBase;

	xMsg3440.Num 		:= 3440;
	xMsg3440.AmmInAdr 	:= iAdrAmmBase2MM;
	xMsg3440.AmmOutAdr 	:= iAdrMM2AmmBase;

	xMsg3441.Num 		:= 3441;
	xMsg3441.AmmInAdr 	:= iAdrAmmBase2MM;
	xMsg3441.AmmOutAdr 	:= iAdrMM2AmmBase;

	xMsg3442.Num 		:= 3442;
	xMsg3442.AmmInAdr 	:= iAdrAmmBase2MM;
	xMsg3442.AmmOutAdr 	:= iAdrMM2AmmBase;

	xMsg3443.Num 		:= 3443;
	xMsg3443.AmmInAdr 	:= iAdrAmmBase2MM;
	xMsg3443.AmmOutAdr 	:= iAdrMM2AmmBase;

	xMsg3446.Num 		:= 3446;
	xMsg3446.AmmInAdr 	:= iAdrAmmBase2MM;
	xMsg3446.AmmOutAdr 	:= iAdrMM2AmmBase;

	xMsg3447.Num 		:= 3447;
	xMsg3447.AmmInAdr 	:= iAdrAmmBase2MM;
	xMsg3447.AmmOutAdr 	:= iAdrMM2AmmBase;

	xMsg3468.Num 		:= 3468;
	xMsg3468.AmmInAdr 	:= iAdrAmmBase2MM;
	xMsg3468.AmmOutAdr 	:= iAdrMM2AmmBase;

	xMsg3516.Num       := 3516;
	xMsg3516.AmmInAdr  := iAdrAmmBase2MM;
	xMsg3516.AmmOutAdr := iAdrMM2AmmBase;

	xMsg3563.Num       := 3563;
	xMsg3563.AmmInAdr  := iAdrAmmBase2MM;
	xMsg3563.AmmOutAdr := iAdrMM2AmmBase;

	xMsg3566.Num       := 3566;
	xMsg3566.AmmInAdr  := iAdrAmmBase2MM;
	xMsg3566.AmmOutAdr := iAdrMM2AmmBase;

	xMsg3573.Num       := 3573;
	xMsg3573.AmmInAdr  := iAdrAmmBase2MM;
	xMsg3573.AmmOutAdr := iAdrMM2AmmBase;

	xMsg9285.Num       := 9285;
	xMsg9285.AmmInAdr  := iAdrAmmBase2MM;
	xMsg9285.AmmOutAdr := iAdrMM2AmmBase;

	xMsg9311.Num       := 9311;
	xMsg9311.AmmInAdr  := iAdrAmmBase2MM;
	xMsg9311.AmmOutAdr := iAdrMM2AmmBase;

	xMsg9351.Num       := 9351;
	xMsg9351.AmmInAdr  := iAdrAmmBase2MM;
	xMsg9351.AmmOutAdr := iAdrMM2AmmBase;

	xMsg9365.Num       := 9365;
	xMsg9365.AmmInAdr  := iAdrAmmBase2MM;
	xMsg9365.AmmOutAdr := iAdrMM2AmmBase;

	xMsg9366.Num       := 9366;
	xMsg9366.AmmInAdr  := iAdrAmmBase2MM;
	xMsg9366.AmmOutAdr := iAdrMM2AmmBase;

	xMsg9367.Num       := 9367;
	xMsg9367.AmmInAdr  := iAdrAmmBase2MM;
	xMsg9367.AmmOutAdr := iAdrMM2AmmBase;

	xMsg9368.Num       := 9368;
	xMsg9368.AmmInAdr  := iAdrAmmBase2MM;
	xMsg9368.AmmOutAdr := iAdrMM2AmmBase;

	xMsg9372.Num       := 9372;
	xMsg9372.AmmInAdr  := iAdrAmmBase2MM;
	xMsg9372.AmmOutAdr := iAdrMM2AmmBase;

END_PROGRAM
```

#### MsgGC.var
```iecst
VAR
	AN_RLSG : BOOL;
	bIASY : BOOL;
	bP_Gen_Reverse : BOOL; (*Reverse power enable -> old name AT24*)
	bP_Reverse_Mon_Ena : BOOL; (*Disable monitoring of reverse power -> old name RLSG_W*)
	bU_Gen_Mon_Ena : BOOL; (*Enable monitoring of generator protection*)
	FG_UASY : BOOL;
	iAdrAmmBase2MM : UDINT;
	iAdrMM2AmmBase : UDINT;
	IASY1_arise : BOOL;
	IASY2_arise : BOOL;
	M_D1400 : BOOL;
	RLSG1_arise : BOOL;
	RLSG2_arise : BOOL;
	STO_IASY : BOOL;
	STO_RLSG : BOOL;
	SY_1m_iasy : BOOL; (*GCB has been closed (ON) for 1 minute*)
	SY_1m_rlsg : BOOL;
	T28 : BOOL; (*Reverse power*)
	xCTD_IASY1 : CTD;
	xCTD_IASY2 : CTD;
	xCTD_RLSG1 : CTD;
	xCTD_RLSG2 : CTD;
	xGR_MAXR_DREHZ : GR_MAXR;
	xGR_MAXR_M_HDREHZ : GR_MAXR;
	xGR_MAX_M_D_1400 : GR_MAXR;
	xGR_MIN_AN_RLSG : GR_MINR;
	xR_TRIG_bIASY : R_TRIG;
	xR_TRIG_T28 : R_TRIG;
	xSR_FG_DIFFUW : SR;
	xTOF_GCB_Off_CNS : TOF;
	xTOF_GCB_Off_RP : TOF;
	xTON_AT24 : TON;
	xTON_Eng_Run_10s : TON;
	xTON_Eng_Run_20s : TON;
	xTON_FG_GENUW : TON;
	xTON_GENREG_F : TON;
	xTON_GSEIN : TON;
	xTP_RLSG_W : TP;
	xTON_T28 : TON;
	xTON_UASY : TON;
	xTON_UASY_Ext : TON;
	xTP_IASY1 : TP;
	xTP_IASY2 : TP;
	xTP_RLSG1 : TP;
	xTP_RLSG2 : TP;
	ZM_GENREG_F : BOOL;
	xR_TRIG_GCB_Off_CNS : R_TRIG;
	xR_TRIG_GCB_Off_RP : R_TRIG;
	xTON_N_EngNom750 : TON;
	xTON_Eng_Run_48s : TON;
	bEng_Run_48s : BOOL;
	xGR_MAX_F_GenBearDE1_Hi : GR_MAXR;
	xGR_MAX_F_GenBearDE2_Hi : GR_MAXR;
	xGR_MAX_F_GenBearNDE1_Hi : GR_MAXR;
	xGR_MAX_F_GenBearNDE2_Hi : GR_MAXR;
	xGR_MAX_F_GenBearDE1_HiHi : GR_MAXR;
	xGR_MAX_F_GenBearDE2_HiHi : GR_MAXR;
	xGR_MAX_F_GenBearNDE1_HiHi : GR_MAXR;
	xGR_MAX_F_GenBearNDE2_HiHi : GR_MAXR;
	xTP_Msg2156 : TP;
	xTP_Msg2157 : TP;
	xTP_Msg2998 : TP;
	xTON2316Set : TON;
	xTON_SecTick : TON;
	xTOF_GenDeexitDem : TOF;
	xTP_gcb_on2dead_bb : TP;
	xMsg1036 : Msg;
	xMsg1037 : Msg;
	xMsg1038 : Msg;
	xMsg1062 : Msg;
	xMsg1073 : Msg;
	xMsg1109 : Msg;
	xMsg1110 : Msg;
	xMsg1111 : Msg;
	xMsg1112 : Msg;
	xMsg1113 : Msg;
	xMsg1121 : Msg;
	xMsg1122 : Msg;
	xMsg1123 : Msg;
	xMsg1124 : Msg;
	xMsg1125 : Msg;
	xMsg1126 : Msg;
	xMsg1127 : Msg;
	xMsg1132 : Msg;
	xMsg1134 : Msg;
	xMsg1143 : Msg;
	xMsg1144 : Msg;
	xMsg1154 : Msg;
	xMsg1155 : Msg;
	xMsg1156 : Msg;
	xMsg1157 : Msg;
	xMsg1158 : Msg;
	xMsg1185 : Msg;
	xMsg2100 : Msg;
	xMsg2105 : Msg;
	xMsg2106 : Msg;
	xMsg2107 : Msg;
	xMsg2108 : Msg;
	xMsg2109 : Msg;
	xMsg2110 : Msg;
	xMsg2115 : Msg;
	xMsg2156 : Msg;
	xMsg2157 : Msg;
	xMsg2202 : Msg;
	xMsg2203 : Msg;
	xMsg2204 : Msg;
	xMsg2205 : Msg;
	xMsg2206 : Msg;
	xMsg2207 : Msg;
	xMsg2208 : Msg; (*A2208 Oilskid tank oil level low *)
	xMsg2277 : Msg;
	xMsg2316 : Msg;
	xMsg2336 : Msg;
	xMsg2371 : Msg; (*A2371 Oil skid Oil flow to DE bearing Low*)
	xMsg2372 : Msg; (*A2372 Oil skid Oil flow to NDE bearing Low*)
	xMsg2373 : Msg; (*A2373 Earth failure generator (MMD) *)
	xMsg2501 : Msg;
	xMsg2502 : Msg;
	xMsg2503 : Msg;
	xMsg2504 : Msg;
	xMsg2505 : Msg; (*W2505 Oilskid low pressure oil filter clogged*)
	xMsg2508 : Msg; (*W2508 Oilskid high pressure oil filter DE clogged*)
	xMsg2555 : Msg;
	xMsg2556 : Msg;
	xMsg2573 : Msg;
	xMsg2631 : Msg;
	xMsg2632 : Msg;
	xMsg2633 : Msg;
	xMsg2634 : Msg;
	xMsg2637 : Msg;
	xMsg2665 : Msg; (*Generator heater circuit breaker tripped*)
	xMsg2690 : Msg;
	xMsg2691 : Msg;
	xMsg2827 : Msg;
	xMsg2828 : Msg;
	xMsg2829 : Msg;
	xMsg2830 : Msg;
	xMsg2998 : Msg;
	xMsg3219 : Msg;
	xMsg3298 : Msg;
	xMsg3299 : Msg;
	xMsg3319 : Msg;
	xMsg3393 : Msg;
	xMsg3418 : Msg; (*W3418 Oilskid oil in oil sump *)
	xMsg3419 : Msg; (*W3419 Oilskid tank oil level measuring signal failure *)
	xMsg3420 : Msg; (*W3420 Oilskid tank oil level low*)
	xMsg3421 : Msg; (*W3421 Oilskid tank oil temperature measuring signal failure*)
	xMsg3422 : Msg; (*W3422 Oilskid tank oil temperature low*)
	xMsg3423 : Msg; (*W3423 Oilskid oil supply temperature measuring signal failure*)
	xMsg3424 : Msg; (*W3424 Oilskid oil supply temperature low*)
	xMsg3425 : Msg; (*W3425 Oilskid oil supply temperature high*)
	xMsg3426 : Msg; (*W3426 Oilskid low pressure oil pump circuit breaker tripped*)
	xMsg3427 : Msg; (*W3427 Oilskid oil flow TO DE bearing measuring signal failure*)
	xMsg3428 : Msg; (*W3428 Oilskid oil flow TO DE bearing low*)
	xMsg3429 : Msg; (*W3429 Oilskid oil flow TO DE bearing high*)
	xMsg3430 : Msg; (*W3430 Oilskid oil flow TO NDE bearing measuring signal failure*)
	xMsg3431 : Msg; (*W3431 Oilskid oil flow TO NDE bearing low*)
	xMsg3432 : Msg; (*W3432 Oilskid oil flow TO NDE bearing high*)
	xMsg3433 : Msg; (*W3433 Oilskid high pressure oil pump circuit breaker tripped*)
	xMsg3434 : Msg; (*W3434 Oilskid high pressure oil pump circuit breaker tripped - UPS*)
	xMsg3435 : Msg; (*W3435 Oilskid oil pressure TO DE bearing measuring signal failure*)
	xMsg3436 : Msg; (*W3436 Oilskid oil pressure TO DE bearing low*)
	xMsg3442 : Msg; (*W3442 Oilskid oil pressure TO NDE bearing measuring signal failure*)
	xMsg3443 : Msg; (*W3443 Oilskid oil pressure TO NDE bearing low*)
	xMsg3446 : Msg; (*W3446 Oilskid high pressure oil filter NDE clogged*)
	xMsg3437 : Msg; (*W3437 Oilskid fan circuit breaker tripped*)
	xMsg3438 : Msg; (*W3438 Oilskid heater circuit breaker tripped*)
	xMsg3439 : Msg; (*W3439 Oilskid main switch auxiliaries opened*)
	xMsg3440 : Msg; (*W3440 Oilskid auxiliaries voltage NOT available*)
	xMsg3441 : Msg; (*W3441 Oilskid auxiliaries voltage NOT available - UPS*)
	xMsg3447 : Msg; (*W3447 Oilskid circulation pump circuit breaker tripped *)
	xMsg3468 : Msg;
	xMsg3516 : Msg;
	xMsg3563 : Msg;
	xMsg3566 : Msg;
	xMsg3573 : Msg;
	xMsg9285 : Msg;
	xMsg9311 : Msg;
	xMsg9351 : Msg;
	xMsg9365 : Msg;
	xMsg9366 : Msg;
	xMsg9367 : Msg;
	xMsg9368 : Msg;
	xMsg9372 : Msg; (*W9372 Earth failure generator (MMD) *)
END_VAR
```

### Program Logical/Generator/ParGC (IEC, version 4.06.0) - + parameter handling

- perm_par.st (not readable text: treated as protected, skipped)
